      global bajada_broca=p[0,0,-0.012,0,0,0]
      $ 661 "bajada≔p[0,0,0.012,0,0,0]"
      global bajada=p[0,0,0.012,0,0,0]
      $ 662 "Direction: Base Z-"
      global move_thread_flag_662=0
      thread move_thread_662():
        enter_critical
        move_thread_flag_662 = 1
        local towardsPos=calculate_point_to_move_towards(p[0.0,0.0,0.0,0.0,0.0,0.0], [0.0,0.0,-1.0], 0.045)
        movel(towardsPos, a=0.025, v=0.02)
        move_thread_flag_662 = 2
        exit_critical
      end
      move_thread_flag_662 = 0
      move_thread_han_662 = run move_thread_662()
      while (True):
        sleep(1.0E-10)
        if (move_thread_flag_662 > 1):
          join move_thread_han_662
          $ 663 "Until (distance)"
          break
        end
        sync()
      end
      $ 664 "Popup: punto contacto alanzdo"
      popup("punto contacto alanzdo", "Mensaje", False, False, blocking=True)
      $ 665 "Direction: Base Z+"
      global move_thread_flag_665=0
      thread move_thread_665():
        enter_critical
        move_thread_flag_665 = 1
        local towardsPos=calculate_point_to_move_towards(p[0.0,0.0,0.0,0.0,0.0,0.0], [0.0,0.0,1.0], 0.001)
        movel(towardsPos, a=0.005, v=0.003)
        move_thread_flag_665 = 2
        exit_critical
      end
      move_thread_flag_665 = 0
      move_thread_han_665 = run move_thread_665()
      while (True):
        sleep(1.0E-10)
        if (move_thread_flag_665 > 1):
          join move_thread_han_665
          $ 666 "Until (distance)"
          break
        end
        sync()
      end
      $ 667 "Wait: 0.3"
      sleep(0.3)
      $ 668 "Set CO[1]=Encender"
      set_configurable_digital_out(1, True)
      $ 669 "Wait: 0.3"
      sleep(0.3)
      $ 670 "Loop 2 times"
      Loop_44 = 0
      while (Loop_44 < 2):
        $ 671 "bajar≔pose_add(get_actual_tcp_pose(), bajada_broca)"
        global bajar= pose_add ( get_actual_tcp_pose (), bajada_broca)
        $ 672 "bajar" "breakAfter"
        movel(bajar, a=0.005, v=0.001)
        $ 673 "subir≔pose_sub(get_actual_tcp_pose(), bajada_broca)"
        global subir= pose_sub ( get_actual_tcp_pose (), bajada_broca)
        $ 674 "subir" "breakAfter"
        movel(subir, a=0.01, v=0.005)
        $ 675 "bajada_broca≔pose_sub(bajada_broca, bajada)"
        global bajada_broca= pose_sub (bajada_broca, bajada)
        Loop_44 = Loop_44 + 1
      end
      $ 676 "Direction: Base Z+"
      global move_thread_flag_676=0
      thread move_thread_676():
        enter_critical
        move_thread_flag_676 = 1
        local towardsPos=calculate_point_to_move_towards(p[0.0,0.0,0.0,0.0,0.0,0.0], [0.0,0.0,1.0], 0.06)
        movel(towardsPos, a=0.035, v=0.03)
        move_thread_flag_676 = 2
        exit_critical
      end
      move_thread_flag_676 = 0
      move_thread_han_676 = run move_thread_676()
      while (True):
        sleep(1.0E-10)
        if (move_thread_flag_676 > 1):
          join move_thread_han_676
          $ 677 "Until (distance)"
          break
        end
        sync()
      end
      $ 678 "Set CO[1]=Apagar"
      set_configurable_digital_out(1, False)
      $ 679 "barreno_actual≔barreno_actual+1"
      global barreno_actual=barreno_actual+1
      $ 680 "If barreno_actual≥barrenos_menos1"
      if (barreno_actual >= barrenos_menos1):
        $ 681 "cambiar_broca≔ True "
        global cambiar_broca=  True
      end
      $ 682 "Call Quitar_broca"
      Quitar_broca()
      $ 683 "Call Poner_broca"
      Poner_broca()
    end
    $ 684 "Popup: Linea2 con full Terminada!"
    popup("Linea2 con full Terminada!", "Mensaje", False, False, blocking=True)
    $ 685 "Posicion3"
    $ 686 "eje7≔3"
    global eje7=3
    $ 687 "Broca_1"
    $ 688 "Linea3"
    $ 689 "Marcar_puntos"
    $ 690 "MoveL"
    $ 691 "Home3" "breakAfter"
    movel(Home3_p, a=0.5, v=0.1)
    $ 692 "Linea3_A" "breakAfter"
    movel(Linea3_A_p, a=0.5, v=0.1)
    $ 693 "Linea3_B" "breakAfter"
    movel(Linea3_B_p, a=0.5, v=0.1)
    $ 694 "Linea3_C" "breakAfter"
    movel(Linea3_C_p, a=0.5, v=0.1)
    $ 695 "Linea3_D" "breakAfter"
    movel(Linea3_D_p, a=0.5, v=0.1)
    $ 696 "Linea3_E" "breakAfter"
    movel(Linea3_E_p, a=0.5, v=0.1)
    $ 697 "Linea3_F" "breakAfter"
    movel(Linea3_F_p, a=0.5, v=0.1)
    $ 698 "AB"
    $ 699 "'desbaste_inicial'"
    # 'desbaste_inicial'
    $ 700 "bajada_broca≔p[0,0,-0.008,0,0,0]"
    global bajada_broca=p[0,0,-0.008,0,0,0]
    $ 701 "barrenos_menos1≔8"
    global barrenos_menos1=8
    $ 702 "barreno_actual≔0"
    global barreno_actual=0
    $ 703 "Loop barreno_actual≤barrenos_menos1"
    while (barreno_actual <= barrenos_menos1):
      $ 704 "Perforacion"
      $ 705 "MoveL"
      $ 706 "internos≔interpolate_pose(Linea3_A, Linea3_B, barreno_actual/barrenos_menos1)"
      global internos= interpolate_pose (Linea3_A_p, Linea3_B_p, barreno_actual/barrenos_menos1)
      $ 707 "internos" "breakAfter"
      movel(internos, a=0.5, v=0.1)
      $ 708 "'desbaste_inicial'"
      # 'desbaste_inicial'
      $ 709 "bajada_broca≔p[0,0,-0.008,0,0,0]"
      global bajada_broca=p[0,0,-0.008,0,0,0]
      $ 710 "bajada≔p[0,0,0.008,0,0,0]"
      global bajada=p[0,0,0.008,0,0,0]
      $ 711 "Direction: Base Z-"
      global move_thread_flag_711=0
      thread move_thread_711():
        enter_critical
        move_thread_flag_711 = 1
        local towardsPos=calculate_point_to_move_towards(p[0.0,0.0,0.0,0.0,0.0,0.0], [0.0,0.0,-1.0], 0.055)
        movel(towardsPos, a=0.015, v=0.02)
        move_thread_flag_711 = 2
        exit_critical
      end
      move_thread_flag_711 = 0
      move_thread_han_711 = run move_thread_711()
      while (True):
        sleep(1.0E-10)
        if (move_thread_flag_711 > 1):
          join move_thread_han_711
          $ 712 "Until (distance)"
          break
        end
        sync()
      end
      $ 713 "Popup: punto contacto alanzdo"
      popup("punto contacto alanzdo", "Mensaje", False, False, blocking=True)
      $ 714 "Direction: Base Z+"
      global move_thread_flag_714=0
      thread move_thread_714():
        enter_critical
        move_thread_flag_714 = 1
        local towardsPos=calculate_point_to_move_towards(p[0.0,0.0,0.0,0.0,0.0,0.0], [0.0,0.0,1.0], 0.002)
        movel(towardsPos, a=0.005, v=0.003)
        move_thread_flag_714 = 2
        exit_critical
      end
      move_thread_flag_714 = 0
      move_thread_han_714 = run move_thread_714()
      while (True):
        sleep(1.0E-10)
        if (move_thread_flag_714 > 1):
          join move_thread_han_714
          $ 715 "Until (distance)"
          break
        end
        sync()
      end
      $ 716 "Wait: 0.3"
      sleep(0.3)
      $ 717 "Set CO[1]=Encender"
      set_configurable_digital_out(1, True)
      $ 718 "Wait: 0.3"
      sleep(0.3)
      $ 719 "Loop 3 times"
      Loop_3 = 0
      while (Loop_3 < 3):
        $ 720 "bajar≔pose_add(get_actual_tcp_pose(), bajada_broca)"
        global bajar= pose_add ( get_actual_tcp_pose (), bajada_broca)
        $ 721 "bajar" "breakAfter"
        movel(bajar, a=0.005, v=0.001)
        $ 722 "subir≔pose_sub(get_actual_tcp_pose(), bajada_broca)"
        global subir= pose_sub ( get_actual_tcp_pose (), bajada_broca)
        $ 723 "subir" "breakAfter"
        movel(subir, a=0.01, v=0.01)
        $ 724 "bajada_broca≔pose_sub(bajada_broca, bajada)"
        global bajada_broca= pose_sub (bajada_broca, bajada)
        Loop_3 = Loop_3 + 1
      end
      $ 725 "Direction: Base Z+"
      global move_thread_flag_725=0
      thread move_thread_725():
        enter_critical
        move_thread_flag_725 = 1
        local towardsPos=calculate_point_to_move_towards(p[0.0,0.0,0.0,0.0,0.0,0.0], [0.0,0.0,1.0], 0.06)
        movel(towardsPos, a=0.035, v=0.03)
        move_thread_flag_725 = 2
        exit_critical
      end
      move_thread_flag_725 = 0
      move_thread_han_725 = run move_thread_725()
      while (True):
        sleep(1.0E-10)
        if (move_thread_flag_725 > 1):
          join move_thread_han_725
          $ 726 "Until (distance)"
          break
        end
        sync()
      end
      $ 727 "Set CO[1]=Apagar"
      set_configurable_digital_out(1, False)
      $ 728 "barreno_actual≔barreno_actual+1"
      global barreno_actual=barreno_actual+1
    end
    $ 731 "CD"
    $ 732 "'desbaste_inicial'"
    # 'desbaste_inicial'
    $ 733 "bajada_broca≔p[0,0,-0.008,0,0,0]"
    global bajada_broca=p[0,0,-0.008,0,0,0]
    $ 734 "barrenos_menos1≔8"
    global barrenos_menos1=8
    $ 735 "barreno_actual≔0"
    global barreno_actual=0
    $ 736 "Loop barreno_actual≤barrenos_menos1"
    while (barreno_actual <= barrenos_menos1):
      $ 737 "Perforacion"
      $ 738 "MoveL"
      $ 739 "internos≔interpolate_pose(Linea3_C, Linea3_D, barreno_actual/barrenos_menos1)"
      global internos= interpolate_pose (Linea3_C_p, Linea3_D_p, barreno_actual/barrenos_menos1)
      $ 740 "internos" "breakAfter"
      movel(internos, a=0.5, v=0.1)
      $ 741 "'desbaste_inicial'"
      # 'desbaste_inicial'
      $ 742 "bajada_broca≔p[0,0,-0.008,0,0,0]"
      global bajada_broca=p[0,0,-0.008,0,0,0]
      $ 743 "bajada≔p[0,0,0.008,0,0,0]"
      global bajada=p[0,0,0.008,0,0,0]
      $ 744 "Direction: Base Z-"
      global move_thread_flag_744=0
      thread move_thread_744():
        enter_critical
        move_thread_flag_744 = 1
        local towardsPos=calculate_point_to_move_towards(p[0.0,0.0,0.0,0.0,0.0,0.0], [0.0,0.0,-1.0], 0.055)
        movel(towardsPos, a=0.015, v=0.02)
        move_thread_flag_744 = 2
        exit_critical
      end
      move_thread_flag_744 = 0
      move_thread_han_744 = run move_thread_744()
      while (True):
        sleep(1.0E-10)
        if (move_thread_flag_744 > 1):
          join move_thread_han_744
          $ 745 "Until (distance)"
          break
        end
        sync()
      end
      $ 746 "Popup: punto contacto alanzdo"
      popup("punto contacto alanzdo", "Mensaje", False, False, blocking=True)
      $ 747 "Direction: Base Z+"
      global move_thread_flag_747=0
      thread move_thread_747():
        enter_critical
        move_thread_flag_747 = 1
        local towardsPos=calculate_point_to_move_towards(p[0.0,0.0,0.0,0.0,0.0,0.0], [0.0,0.0,1.0], 0.002)
        movel(towardsPos, a=0.005, v=0.003)
        move_thread_flag_747 = 2
        exit_critical
      end
      move_thread_flag_747 = 0
      move_thread_han_747 = run move_thread_747()
      while (True):
        sleep(1.0E-10)
        if (move_thread_flag_747 > 1):
          join move_thread_han_747
          $ 748 "Until (distance)"
          break
        end
        sync()
      end
      $ 749 "Wait: 0.3"
      sleep(0.3)
      $ 750 "Set CO[1]=Encender"
      set_configurable_digital_out(1, True)
      $ 751 "Wait: 0.3"
      sleep(0.3)
      $ 752 "Loop 3 times"
      Loop_6 = 0
      while (Loop_6 < 3):
        $ 753 "bajar≔pose_add(get_actual_tcp_pose(), bajada_broca)"
        global bajar= pose_add ( get_actual_tcp_pose (), bajada_broca)
        $ 754 "bajar" "breakAfter"
        movel(bajar, a=0.005, v=0.001)
        $ 755 "subir≔pose_sub(get_actual_tcp_pose(), bajada_broca)"
        global subir= pose_sub ( get_actual_tcp_pose (), bajada_broca)
        $ 756 "subir" "breakAfter"
        movel(subir, a=0.01, v=0.01)
        $ 757 "bajada_broca≔pose_sub(bajada_broca, bajada)"
        global bajada_broca= pose_sub (bajada_broca, bajada)
        Loop_6 = Loop_6 + 1
      end
      $ 758 "Direction: Base Z+"
      global move_thread_flag_758=0
      thread move_thread_758():
        enter_critical
        move_thread_flag_758 = 1
        local towardsPos=calculate_point_to_move_towards(p[0.0,0.0,0.0,0.0,0.0,0.0], [0.0,0.0,1.0], 0.06)
        movel(towardsPos, a=0.035, v=0.03)
        move_thread_flag_758 = 2
        exit_critical
      end
      move_thread_flag_758 = 0
      move_thread_han_758 = run move_thread_758()
      while (True):
        sleep(1.0E-10)
        if (move_thread_flag_758 > 1):
          join move_thread_han_758
          $ 759 "Until (distance)"
          break
        end
        sync()
      end
      $ 760 "Set CO[1]=Apagar"
      set_configurable_digital_out(1, False)
      $ 761 "barreno_actual≔barreno_actual+1"
      global barreno_actual=barreno_actual+1
    end
    $ 764 "EF"
    $ 765 "'desbaste_inicial'"
    # 'desbaste_inicial'
    $ 766 "bajada_broca≔p[0,0,-0.008,0,0,0]"
    global bajada_broca=p[0,0,-0.008,0,0,0]
    $ 767 "barrenos_menos1≔8"
    global barrenos_menos1=8
    $ 768 "barreno_actual≔0"
    global barreno_actual=0
    $ 769 "Loop barreno_actual≤barrenos_menos1"
    while (barreno_actual <= barrenos_menos1):
      $ 770 "Perforacion"
      $ 771 "MoveL"
      $ 772 "internos≔interpolate_pose(Linea3_E, Linea3_F, barreno_actual/barrenos_menos1)"
      global internos= interpolate_pose (Linea3_E_p, Linea3_F_p, barreno_actual/barrenos_menos1)
      $ 773 "internos" "breakAfter"
      movel(internos, a=0.5, v=0.1)
      $ 774 "'desbaste_inicial'"
      # 'desbaste_inicial'
      $ 775 "bajada_broca≔p[0,0,-0.008,0,0,0]"
      global bajada_broca=p[0,0,-0.008,0,0,0]
      $ 776 "bajada≔p[0,0,0.008,0,0,0]"
      global bajada=p[0,0,0.008,0,0,0]
      $ 777 "Direction: Base Z-"
      global move_thread_flag_777=0
      thread move_thread_777():
        enter_critical
        move_thread_flag_777 = 1
        local towardsPos=calculate_point_to_move_towards(p[0.0,0.0,0.0,0.0,0.0,0.0], [0.0,0.0,-1.0], 0.055)
        movel(towardsPos, a=0.015, v=0.02)
        move_thread_flag_777 = 2
        exit_critical
      end
      move_thread_flag_777 = 0
      move_thread_han_777 = run move_thread_777()
      while (True):
        sleep(1.0E-10)
        if (move_thread_flag_777 > 1):
          join move_thread_han_777
          $ 778 "Until (distance)"
          break
        end
        sync()
      end
      $ 779 "Popup: punto contacto alanzdo"
      popup("punto contacto alanzdo", "Mensaje", False, False, blocking=True)
      $ 780 "Direction: Base Z+"
      global move_thread_flag_780=0
      thread move_thread_780():
        enter_critical
        move_thread_flag_780 = 1
        local towardsPos=calculate_point_to_move_towards(p[0.0,0.0,0.0,0.0,0.0,0.0], [0.0,0.0,1.0], 0.002)
        movel(towardsPos, a=0.005, v=0.003)
        move_thread_flag_780 = 2
        exit_critical
      end
      move_thread_flag_780 = 0
      move_thread_han_780 = run move_thread_780()
      while (True):
        sleep(1.0E-10)
        if (move_thread_flag_780 > 1):
          join move_thread_han_780
          $ 781 "Until (distance)"
          break
        end
        sync()
      end
      $ 782 "Wait: 0.3"
      sleep(0.3)
      $ 783 "Set CO[1]=Encender"
      set_configurable_digital_out(1, True)
      $ 784 "Wait: 0.3"
      sleep(0.3)
      $ 785 "Loop 3 times"
      Loop_8 = 0
      while (Loop_8 < 3):
        $ 786 "bajar≔pose_add(get_actual_tcp_pose(), bajada_broca)"
        global bajar= pose_add ( get_actual_tcp_pose (), bajada_broca)
        $ 787 "bajar" "breakAfter"
        movel(bajar, a=0.005, v=0.001)
        $ 788 "subir≔pose_sub(get_actual_tcp_pose(), bajada_broca)"
        global subir= pose_sub ( get_actual_tcp_pose (), bajada_broca)
        $ 789 "subir" "breakAfter"
        movel(subir, a=0.01, v=0.01)
        $ 790 "bajada_broca≔pose_sub(bajada_broca, bajada)"
        global bajada_broca= pose_sub (bajada_broca, bajada)
        Loop_8 = Loop_8 + 1
      end
      $ 791 "Direction: Base Z+"
      global move_thread_flag_791=0
      thread move_thread_791():
        enter_critical
        move_thread_flag_791 = 1
        local towardsPos=calculate_point_to_move_towards(p[0.0,0.0,0.0,0.0,0.0,0.0], [0.0,0.0,1.0], 0.06)
        movel(towardsPos, a=0.035, v=0.03)
        move_thread_flag_791 = 2
        exit_critical
      end
      move_thread_flag_791 = 0
      move_thread_han_791 = run move_thread_791()
      while (True):
        sleep(1.0E-10)
        if (move_thread_flag_791 > 1):
          join move_thread_han_791
          $ 792 "Until (distance)"
          break
        end
        sync()
      end
      $ 793 "Set CO[1]=Apagar"
      set_configurable_digital_out(1, False)
      $ 794 "barreno_actual≔barreno_actual+1"
      global barreno_actual=barreno_actual+1
    end
    $ 797 "Popup: Linea3 con chica Terminada!"
    popup("Linea3 con chica Terminada!", "Mensaje", False, False, blocking=True)
    $ 798 "Linea4"
    $ 799 "Marcar_puntos"
    $ 800 "MoveL"
    $ 801 "Home3" "breakAfter"
    movel(Home3_p, a=0.5, v=0.1)
    $ 802 "Linea4_A" "breakAfter"
    movel(Linea4_A_p, a=0.5, v=0.1)
    $ 803 "Linea4_B" "breakAfter"
    movel(Linea4_B_p, a=0.5, v=0.1)
    $ 804 "Linea4_C" "breakAfter"
    movel(Linea4_C_p, a=0.5, v=0.1)
    $ 805 "Linea4_D" "breakAfter"
    movel(Linea4_D_p, a=0.5, v=0.1)
    $ 806 "Linea4_E" "breakAfter"
    movel(Linea4_E_p, a=0.5, v=0.1)
    $ 807 "Linea4_F" "breakAfter"
    movel(Linea4_F_p, a=0.5, v=0.1)
    $ 808 "AB"
    $ 809 "'desbaste_inicial'"
    # 'desbaste_inicial'
    $ 810 "bajada_broca≔p[0,0,-0.008,0,0,0]"
    global bajada_broca=p[0,0,-0.008,0,0,0]
    $ 811 "barrenos_menos1≔8"
    global barrenos_menos1=8
    $ 812 "barreno_actual≔0"
    global barreno_actual=0
    $ 813 "Loop barreno_actual≤barrenos_menos1"
    while (barreno_actual <= barrenos_menos1):
      $ 814 "Perforacion"
      $ 815 "MoveL"
      $ 816 "internos≔interpolate_pose(Linea4_A, Linea4_B, barreno_actual/barrenos_menos1)"
      global internos= interpolate_pose (Linea4_A_p, Linea4_B_p, barreno_actual/barrenos_menos1)
      $ 817 "internos" "breakAfter"
      movel(internos, a=0.5, v=0.1)
      $ 818 "'desbaste_inicial'"
      # 'desbaste_inicial'
      $ 819 "bajada_broca≔p[0,0,-0.008,0,0,0]"
      global bajada_broca=p[0,0,-0.008,0,0,0]
      $ 820 "bajada≔p[0,0,0.008,0,0,0]"
      global bajada=p[0,0,0.008,0,0,0]
      $ 821 "Direction: Base Z-"
      global move_thread_flag_821=0
      thread move_thread_821():
        enter_critical
        move_thread_flag_821 = 1
        local towardsPos=calculate_point_to_move_towards(p[0.0,0.0,0.0,0.0,0.0,0.0], [0.0,0.0,-1.0], 0.055)
        movel(towardsPos, a=0.015, v=0.02)
        move_thread_flag_821 = 2
        exit_critical
      end
      move_thread_flag_821 = 0
      move_thread_han_821 = run move_thread_821()
      while (True):
        sleep(1.0E-10)
        if (move_thread_flag_821 > 1):
          join move_thread_han_821
          $ 822 "Until (distance)"
          break
        end
        sync()
      end
      $ 823 "Popup: punto contacto alanzdo"
      popup("punto contacto alanzdo", "Mensaje", False, False, blocking=True)
      $ 824 "Direction: Base Z+"
      global move_thread_flag_824=0
      thread move_thread_824():
        enter_critical
        move_thread_flag_824 = 1
        local towardsPos=calculate_point_to_move_towards(p[0.0,0.0,0.0,0.0,0.0,0.0], [0.0,0.0,1.0], 0.002)
        movel(towardsPos, a=0.005, v=0.003)
        move_thread_flag_824 = 2
        exit_critical
      end
      move_thread_flag_824 = 0
      move_thread_han_824 = run move_thread_824()
      while (True):
        sleep(1.0E-10)
        if (move_thread_flag_824 > 1):
          join move_thread_han_824
          $ 825 "Until (distance)"
          break
        end
        sync()
      end
      $ 826 "Wait: 0.3"
      sleep(0.3)
      $ 827 "Set CO[1]=Encender"
      set_configurable_digital_out(1, True)
      $ 828 "Wait: 0.3"
      sleep(0.3)
      $ 829 "Loop 3 times"
      Loop_12 = 0
      while (Loop_12 < 3):
        $ 830 "bajar≔pose_add(get_actual_tcp_pose(), bajada_broca)"
        global bajar= pose_add ( get_actual_tcp_pose (), bajada_broca)
        $ 831 "bajar" "breakAfter"
        movel(bajar, a=0.005, v=0.001)
        $ 832 "subir≔pose_sub(get_actual_tcp_pose(), bajada_broca)"
        global subir= pose_sub ( get_actual_tcp_pose (), bajada_broca)
        $ 833 "subir" "breakAfter"
        movel(subir, a=0.01, v=0.01)
        $ 834 "bajada_broca≔pose_sub(bajada_broca, bajada)"
        global bajada_broca= pose_sub (bajada_broca, bajada)
        Loop_12 = Loop_12 + 1
      end
      $ 835 "Direction: Base Z+"
      global move_thread_flag_835=0
      thread move_thread_835():
        enter_critical
        move_thread_flag_835 = 1
        local towardsPos=calculate_point_to_move_towards(p[0.0,0.0,0.0,0.0,0.0,0.0], [0.0,0.0,1.0], 0.06)
        movel(towardsPos, a=0.035, v=0.03)
        move_thread_flag_835 = 2
        exit_critical
      end
      move_thread_flag_835 = 0
      move_thread_han_835 = run move_thread_835()
      while (True):
        sleep(1.0E-10)
        if (move_thread_flag_835 > 1):
          join move_thread_han_835
          $ 836 "Until (distance)"
          break
        end
        sync()
      end
      $ 837 "Set CO[1]=Apagar"
      set_configurable_digital_out(1, False)
      $ 838 "barreno_actual≔barreno_actual+1"
      global barreno_actual=barreno_actual+1
    end
    $ 841 "CD"
    $ 842 "'desbaste_inicial'"
    # 'desbaste_inicial'
    $ 843 "bajada_broca≔p[0,0,-0.008,0,0,0]"
    global bajada_broca=p[0,0,-0.008,0,0,0]
    $ 844 "barrenos_menos1≔8"
    global barrenos_menos1=8
    $ 845 "barreno_actual≔0"
    global barreno_actual=0
    $ 846 "Loop barreno_actual≤barrenos_menos1"
    while (barreno_actual <= barrenos_menos1):
      $ 847 "Perforacion"
      $ 848 "MoveL"
      $ 849 "internos≔interpolate_pose(Linea4_C, Linea4_D, barreno_actual/barrenos_menos1)"
      global internos= interpolate_pose (Linea4_C_p, Linea4_D_p, barreno_actual/barrenos_menos1)
      $ 850 "internos" "breakAfter"
      movel(internos, a=0.5, v=0.1)
      $ 851 "'desbaste_inicial'"
      # 'desbaste_inicial'
      $ 852 "bajada_broca≔p[0,0,-0.008,0,0,0]"
      global bajada_broca=p[0,0,-0.008,0,0,0]
      $ 853 "bajada≔p[0,0,0.008,0,0,0]"
      global bajada=p[0,0,0.008,0,0,0]
      $ 854 "Direction: Base Z-"
      global move_thread_flag_854=0
      thread move_thread_854():
        enter_critical
        move_thread_flag_854 = 1
        local towardsPos=calculate_point_to_move_towards(p[0.0,0.0,0.0,0.0,0.0,0.0], [0.0,0.0,-1.0], 0.055)
        movel(towardsPos, a=0.015, v=0.02)
        move_thread_flag_854 = 2
        exit_critical
      end
      move_thread_flag_854 = 0
      move_thread_han_854 = run move_thread_854()
      while (True):
        sleep(1.0E-10)
        if (move_thread_flag_854 > 1):
          join move_thread_han_854
          $ 855 "Until (distance)"
          break
        end
        sync()
      end
      $ 856 "Popup: punto contacto alanzdo"
      popup("punto contacto alanzdo", "Mensaje", False, False, blocking=True)
      $ 857 "Direction: Base Z+"
      global move_thread_flag_857=0
      thread move_thread_857():
        enter_critical
        move_thread_flag_857 = 1
        local towardsPos=calculate_point_to_move_towards(p[0.0,0.0,0.0,0.0,0.0,0.0], [0.0,0.0,1.0], 0.002)
        movel(towardsPos, a=0.005, v=0.003)
        move_thread_flag_857 = 2
        exit_critical
      end
      move_thread_flag_857 = 0
      move_thread_han_857 = run move_thread_857()
      while (True):
        sleep(1.0E-10)
        if (move_thread_flag_857 > 1):
          join move_thread_han_857
          $ 858 "Until (distance)"
          break
        end
        sync()
      end
      $ 859 "Wait: 0.3"
      sleep(0.3)
      $ 860 "Set CO[1]=Encender"
      set_configurable_digital_out(1, True)
      $ 861 "Wait: 0.3"
      sleep(0.3)
      $ 862 "Loop 3 times"
      Loop_15 = 0
      while (Loop_15 < 3):
        $ 863 "bajar≔pose_add(get_actual_tcp_pose(), bajada_broca)"
        global bajar= pose_add ( get_actual_tcp_pose (), bajada_broca)
        $ 864 "bajar" "breakAfter"
        movel(bajar, a=0.005, v=0.001)
        $ 865 "subir≔pose_sub(get_actual_tcp_pose(), bajada_broca)"
        global subir= pose_sub ( get_actual_tcp_pose (), bajada_broca)
        $ 866 "subir" "breakAfter"
        movel(subir, a=0.01, v=0.01)
        $ 867 "bajada_broca≔pose_sub(bajada_broca, bajada)"
        global bajada_broca= pose_sub (bajada_broca, bajada)
        Loop_15 = Loop_15 + 1
      end
      $ 868 "Direction: Base Z+"
      global move_thread_flag_868=0
      thread move_thread_868():
        enter_critical
        move_thread_flag_868 = 1
        local towardsPos=calculate_point_to_move_towards(p[0.0,0.0,0.0,0.0,0.0,0.0], [0.0,0.0,1.0], 0.06)
        movel(towardsPos, a=0.035, v=0.03)
        move_thread_flag_868 = 2
        exit_critical
      end
      move_thread_flag_868 = 0
      move_thread_han_868 = run move_thread_868()
      while (True):
        sleep(1.0E-10)
        if (move_thread_flag_868 > 1):
          join move_thread_han_868
          $ 869 "Until (distance)"
          break
        end
        sync()
      end
      $ 870 "Set CO[1]=Apagar"
      set_configurable_digital_out(1, False)
      $ 871 "barreno_actual≔barreno_actual+1"
      global barreno_actual=barreno_actual+1
    end
    $ 874 "EF"
    $ 875 "'desbaste_inicial'"
    # 'desbaste_inicial'
    $ 876 "bajada_broca≔p[0,0,-0.008,0,0,0]"
    global bajada_broca=p[0,0,-0.008,0,0,0]
    $ 877 "barrenos_menos1≔8"
    global barrenos_menos1=8
    $ 878 "barreno_actual≔0"
    global barreno_actual=0
    $ 879 "Loop barreno_actual≤barrenos_menos1"
    while (barreno_actual <= barrenos_menos1):
      $ 880 "Perforacion"
      $ 881 "MoveL"
      $ 882 "internos≔interpolate_pose(Linea4_E, Linea4_F, barreno_actual/barrenos_menos1)"
      global internos= interpolate_pose (Linea4_E_p, Linea4_F_p, barreno_actual/barrenos_menos1)
      $ 883 "internos" "breakAfter"
      movel(internos, a=0.5, v=0.1)
      $ 884 "'desbaste_inicial'"
      # 'desbaste_inicial'
      $ 885 "bajada_broca≔p[0,0,-0.008,0,0,0]"
      global bajada_broca=p[0,0,-0.008,0,0,0]
      $ 886 "bajada≔p[0,0,0.008,0,0,0]"
      global bajada=p[0,0,0.008,0,0,0]
      $ 887 "Direction: Base Z-"
      global move_thread_flag_887=0
      thread move_thread_887():
        enter_critical
        move_thread_flag_887 = 1
        local towardsPos=calculate_point_to_move_towards(p[0.0,0.0,0.0,0.0,0.0,0.0], [0.0,0.0,-1.0], 0.055)
        movel(towardsPos, a=0.015, v=0.02)
        move_thread_flag_887 = 2
        exit_critical
      end
      move_thread_flag_887 = 0
      move_thread_han_887 = run move_thread_887()
      while (True):
        sleep(1.0E-10)
        if (move_thread_flag_887 > 1):
          join move_thread_han_887
          $ 888 "Until (distance)"
          break
        end
        sync()
      end
      $ 889 "Popup: punto contacto alanzdo"
      popup("punto contacto alanzdo", "Mensaje", False, False, blocking=True)
      $ 890 "Direction: Base Z+"
      global move_thread_flag_890=0
      thread move_thread_890():
        enter_critical
        move_thread_flag_890 = 1
        local towardsPos=calculate_point_to_move_towards(p[0.0,0.0,0.0,0.0,0.0,0.0], [0.0,0.0,1.0], 0.002)
        movel(towardsPos, a=0.005, v=0.003)
        move_thread_flag_890 = 2
        exit_critical
      end
      move_thread_flag_890 = 0
      move_thread_han_890 = run move_thread_890()
      while (True):
        sleep(1.0E-10)
        if (move_thread_flag_890 > 1):
          join move_thread_han_890
          $ 891 "Until (distance)"
          break
        end
        sync()
      end
      $ 892 "Wait: 0.3"
      sleep(0.3)
      $ 893 "Set CO[1]=Encender"
      set_configurable_digital_out(1, True)
      $ 894 "Wait: 0.3"
      sleep(0.3)
      $ 895 "Loop 3 times"
      Loop_19 = 0
      while (Loop_19 < 3):
        $ 896 "bajar≔pose_add(get_actual_tcp_pose(), bajada_broca)"
        global bajar= pose_add ( get_actual_tcp_pose (), bajada_broca)
        $ 897 "bajar" "breakAfter"
        movel(bajar, a=0.005, v=0.001)
        $ 898 "subir≔pose_sub(get_actual_tcp_pose(), bajada_broca)"
        global subir= pose_sub ( get_actual_tcp_pose (), bajada_broca)
        $ 899 "subir" "breakAfter"
        movel(subir, a=0.01, v=0.01)
        $ 900 "bajada_broca≔pose_sub(bajada_broca, bajada)"
        global bajada_broca= pose_sub (bajada_broca, bajada)
        Loop_19 = Loop_19 + 1
      end
      $ 901 "Direction: Base Z+"
      global move_thread_flag_901=0
      thread move_thread_901():
        enter_critical
        move_thread_flag_901 = 1
        local towardsPos=calculate_point_to_move_towards(p[0.0,0.0,0.0,0.0,0.0,0.0], [0.0,0.0,1.0], 0.06)
        movel(towardsPos, a=0.035, v=0.03)
        move_thread_flag_901 = 2
        exit_critical
      end
      move_thread_flag_901 = 0
      move_thread_han_901 = run move_thread_901()
      while (True):
        sleep(1.0E-10)
        if (move_thread_flag_901 > 1):
          join move_thread_han_901
          $ 902 "Until (distance)"
          break
        end
        sync()
      end
      $ 903 "Set CO[1]=Apagar"
      set_configurable_digital_out(1, False)
      $ 904 "barreno_actual≔barreno_actual+1"
      global barreno_actual=barreno_actual+1
      $ 905 "If barreno_actual≥barrenos_menos1"
      if (barreno_actual >= barrenos_menos1):
        $ 906 "cambiar_broca≔ True "
        global cambiar_broca=  True
      end
    end
    $ 909 "Popup: Linea4 con chica Terminada!"
    popup("Linea4 con chica Terminada!", "Mensaje", False, False, blocking=True)
    $ 910 "Broca_2"
    $ 911 "Linea3"
    $ 912 "Marcar_puntos"
    $ 913 "MoveL"
    $ 914 "Home3" "breakAfter"
    movel(Home3_p, a=0.5, v=0.1)
    $ 915 "Linea3_A" "breakAfter"
    movel(Linea3_A_p, a=0.5, v=0.1)
    $ 916 "Linea3_B" "breakAfter"
    movel(Linea3_B_p, a=0.5, v=0.1)
    $ 917 "Linea3_C" "breakAfter"
    movel(Linea3_C_p, a=0.5, v=0.1)
    $ 918 "Linea3_D" "breakAfter"
    movel(Linea3_D_p, a=0.5, v=0.1)
    $ 919 "Linea3_E" "breakAfter"
    movel(Linea3_E_p, a=0.5, v=0.1)
    $ 920 "Linea3_F" "breakAfter"
    movel(Linea3_F_p, a=0.5, v=0.1)
    $ 921 "AB"
    $ 922 "'desbaste_inicial'"
    # 'desbaste_inicial'
    $ 923 "bajada_broca≔p[0,0,-0.012,0,0,0]"
    global bajada_broca=p[0,0,-0.012,0,0,0]
    $ 924 "barrenos_menos1≔8"
    global barrenos_menos1=8
    $ 925 "barreno_actual≔0"
    global barreno_actual=0
    $ 926 "Loop barreno_actual≤barrenos_menos1"
    while (barreno_actual <= barrenos_menos1):
      $ 927 "Perforacion"
      $ 928 "MoveL"
      $ 929 "internos≔interpolate_pose(Linea3_A, Linea3_B, barreno_actual/barrenos_menos1)"
      global internos= interpolate_pose (Linea3_A_p, Linea3_B_p, barreno_actual/barrenos_menos1)
      $ 930 "internos" "breakAfter"
      movel(internos, a=0.5, v=0.1)
      $ 931 "'desbaste_inicial'"
      # 'desbaste_inicial'
      $ 932 "bajada_broca≔p[0,0,-0.012,0,0,0]"
      global bajada_broca=p[0,0,-0.012,0,0,0]
      $ 933 "bajada≔p[0,0,0.012,0,0,0]"
      global bajada=p[0,0,0.012,0,0,0]
      $ 934 "Direction: Base Z-"
      global move_thread_flag_934=0
      thread move_thread_934():
        enter_critical
        move_thread_flag_934 = 1
        local towardsPos=calculate_point_to_move_towards(p[0.0,0.0,0.0,0.0,0.0,0.0], [0.0,0.0,-1.0], 0.055)
        movel(towardsPos, a=0.015, v=0.02)
        move_thread_flag_934 = 2
        exit_critical
      end
      move_thread_flag_934 = 0
      move_thread_han_934 = run move_thread_934()
      while (True):
        sleep(1.0E-10)
        if (move_thread_flag_934 > 1):
          join move_thread_han_934
          $ 935 "Until (distance)"
          break
        end
        sync()
      end
      $ 936 "Popup: punto contacto alanzdo"
      popup("punto contacto alanzdo", "Mensaje", False, False, blocking=True)
      $ 937 "Direction: Base Z+"
      global move_thread_flag_937=0
      thread move_thread_937():
        enter_critical
        move_thread_flag_937 = 1
        local towardsPos=calculate_point_to_move_towards(p[0.0,0.0,0.0,0.0,0.0,0.0], [0.0,0.0,1.0], 0.001)
        movel(towardsPos, a=0.005, v=0.003)
        move_thread_flag_937 = 2
        exit_critical
      end
      move_thread_flag_937 = 0
      move_thread_han_937 = run move_thread_937()
      while (True):
        sleep(1.0E-10)
        if (move_thread_flag_937 > 1):
          join move_thread_han_937
          $ 938 "Until (distance)"
          break
        end
        sync()
      end
      $ 939 "Wait: 0.3"
      sleep(0.3)
      $ 940 "Set CO[1]=Encender"
      set_configurable_digital_out(1, True)
      $ 941 "Wait: 0.3"
      sleep(0.3)
      $ 942 "Loop 2 times"
      Loop_23 = 0
      while (Loop_23 < 2):
        $ 943 "bajar≔pose_add(get_actual_tcp_pose(), bajada_broca)"
        global bajar= pose_add ( get_actual_tcp_pose (), bajada_broca)
        $ 944 "bajar" "breakAfter"
        movel(bajar, a=0.005, v=0.001)
        $ 945 "subir≔pose_sub(get_actual_tcp_pose(), bajada_broca)"
        global subir= pose_sub ( get_actual_tcp_pose (), bajada_broca)
        $ 946 "subir" "breakAfter"
        movel(subir, a=0.01, v=0.01)
        $ 947 "bajada_broca≔pose_sub(bajada_broca, bajada)"
        global bajada_broca= pose_sub (bajada_broca, bajada)
        Loop_23 = Loop_23 + 1
      end
      $ 948 "Direction: Base Z+"
      global move_thread_flag_948=0
      thread move_thread_948():
        enter_critical
        move_thread_flag_948 = 1
        local towardsPos=calculate_point_to_move_towards(p[0.0,0.0,0.0,0.0,0.0,0.0], [0.0,0.0,1.0], 0.06)
        movel(towardsPos, a=0.035, v=0.03)
        move_thread_flag_948 = 2
        exit_critical
      end
      move_thread_flag_948 = 0
      move_thread_han_948 = run move_thread_948()
      while (True):
        sleep(1.0E-10)
        if (move_thread_flag_948 > 1):
          join move_thread_han_948
          $ 949 "Until (distance)"
          break
        end
        sync()
      end
      $ 950 "Set CO[1]=Apagar"
      set_configurable_digital_out(1, False)
      $ 951 "barreno_actual≔barreno_actual+1"
      global barreno_actual=barreno_actual+1
    end
    $ 954 "CD"
    $ 955 "'desbaste_inicial'"
    # 'desbaste_inicial'
    $ 956 "bajada_broca≔p[0,0,-0.012,0,0,0]"
    global bajada_broca=p[0,0,-0.012,0,0,0]
    $ 957 "barrenos_menos1≔8"
    global barrenos_menos1=8
    $ 958 "barreno_actual≔0"
    global barreno_actual=0
    $ 959 "Loop barreno_actual≤barrenos_menos1"
    while (barreno_actual <= barrenos_menos1):
      $ 960 "Perforacion"
      $ 961 "MoveL"
      $ 962 "internos≔interpolate_pose(Linea3_C, Linea3_D, barreno_actual/barrenos_menos1)"
      global internos= interpolate_pose (Linea3_C_p, Linea3_D_p, barreno_actual/barrenos_menos1)
      $ 963 "internos" "breakAfter"
      movel(internos, a=0.5, v=0.1)
      $ 964 "'desbaste_inicial'"
      # 'desbaste_inicial'
      $ 965 "bajada_broca≔p[0,0,-0.012,0,0,0]"
      global bajada_broca=p[0,0,-0.012,0,0,0]
      $ 966 "bajada≔p[0,0,0.012,0,0,0]"
      global bajada=p[0,0,0.012,0,0,0]
      $ 967 "Direction: Base Z-"
      global move_thread_flag_967=0
      thread move_thread_967():
        enter_critical
        move_thread_flag_967 = 1
        local towardsPos=calculate_point_to_move_towards(p[0.0,0.0,0.0,0.0,0.0,0.0], [0.0,0.0,-1.0], 0.055)
        movel(towardsPos, a=0.015, v=0.02)
        move_thread_flag_967 = 2
        exit_critical
      end
      move_thread_flag_967 = 0
      move_thread_han_967 = run move_thread_967()
      while (True):
        sleep(1.0E-10)
        if (move_thread_flag_967 > 1):
          join move_thread_han_967
          $ 968 "Until (distance)"
          break
        end
        sync()
      end
      $ 969 "Popup: punto contacto alanzdo"
      popup("punto contacto alanzdo", "Mensaje", False, False, blocking=True)
      $ 970 "Direction: Base Z+"
      global move_thread_flag_970=0
      thread move_thread_970():
        enter_critical
        move_thread_flag_970 = 1
        local towardsPos=calculate_point_to_move_towards(p[0.0,0.0,0.0,0.0,0.0,0.0], [0.0,0.0,1.0], 0.001)
        movel(towardsPos, a=0.005, v=0.003)
        move_thread_flag_970 = 2
        exit_critical
      end
      move_thread_flag_970 = 0
      move_thread_han_970 = run move_thread_970()
      while (True):
        sleep(1.0E-10)
        if (move_thread_flag_970 > 1):
          join move_thread_han_970
          $ 971 "Until (distance)"
          break
        end
        sync()
      end
      $ 972 "Wait: 0.3"
      sleep(0.3)
      $ 973 "Set CO[1]=Encender"
      set_configurable_digital_out(1, True)
      $ 974 "Wait: 0.3"
      sleep(0.3)
      $ 975 "Loop 2 times"
      Loop_25 = 0
      while (Loop_25 < 2):
        $ 976 "bajar≔pose_add(get_actual_tcp_pose(), bajada_broca)"
        global bajar= pose_add ( get_actual_tcp_pose (), bajada_broca)
        $ 977 "bajar" "breakAfter"
        movel(bajar, a=0.005, v=0.001)
        $ 978 "subir≔pose_sub(get_actual_tcp_pose(), bajada_broca)"
        global subir= pose_sub ( get_actual_tcp_pose (), bajada_broca)
        $ 979 "subir" "breakAfter"
        movel(subir, a=0.01, v=0.01)
        $ 980 "bajada_broca≔pose_sub(bajada_broca, bajada)"
        global bajada_broca= pose_sub (bajada_broca, bajada)
        Loop_25 = Loop_25 + 1
      end
      $ 981 "Direction: Base Z+"
      global move_thread_flag_981=0
      thread move_thread_981():
        enter_critical
        move_thread_flag_981 = 1
        local towardsPos=calculate_point_to_move_towards(p[0.0,0.0,0.0,0.0,0.0,0.0], [0.0,0.0,1.0], 0.06)
        movel(towardsPos, a=0.035, v=0.03)
        move_thread_flag_981 = 2
        exit_critical
      end
      move_thread_flag_981 = 0
      move_thread_han_981 = run move_thread_981()
      while (True):
        sleep(1.0E-10)
        if (move_thread_flag_981 > 1):
          join move_thread_han_981
          $ 982 "Until (distance)"
          break
        end
        sync()
      end
      $ 983 "Set CO[1]=Apagar"
      set_configurable_digital_out(1, False)
      $ 984 "barreno_actual≔barreno_actual+1"
      global barreno_actual=barreno_actual+1
    end
    $ 987 "EF"
    $ 988 "'desbaste_inicial'"
    # 'desbaste_inicial'
    $ 989 "bajada_broca≔p[0,0,-0.012,0,0,0]"
    global bajada_broca=p[0,0,-0.012,0,0,0]
    $ 990 "barrenos_menos1≔8"
    global barrenos_menos1=8
    $ 991 "barreno_actual≔0"
    global barreno_actual=0
    $ 992 "Loop barreno_actual≤barrenos_menos1"
    while (barreno_actual <= barrenos_menos1):
      $ 993 "Perforacion"
      $ 994 "MoveL"
      $ 995 "internos≔interpolate_pose(Linea3_E, Linea3_F, barreno_actual/barrenos_menos1)"
      global internos= interpolate_pose (Linea3_E_p, Linea3_F_p, barreno_actual/barrenos_menos1)
      $ 996 "internos" "breakAfter"
      movel(internos, a=0.5, v=0.1)
      $ 997 "'desbaste_inicial'"
      # 'desbaste_inicial'
      $ 998 "bajada_broca≔p[0,0,-0.012,0,0,0]"
      global bajada_broca=p[0,0,-0.012,0,0,0]
      $ 999 "bajada≔p[0,0,0.012,0,0,0]"
      global bajada=p[0,0,0.012,0,0,0]
      $ 1000 "Direction: Base Z-"
      global move_thread_flag_1000=0
      thread move_thread_1000():
        enter_critical
        move_thread_flag_1000 = 1
        local towardsPos=calculate_point_to_move_towards(p[0.0,0.0,0.0,0.0,0.0,0.0], [0.0,0.0,-1.0], 0.055)
        movel(towardsPos, a=0.015, v=0.02)
        move_thread_flag_1000 = 2
        exit_critical
      end
      move_thread_flag_1000 = 0
      move_thread_han_1000 = run move_thread_1000()
      while (True):
        sleep(1.0E-10)
        if (move_thread_flag_1000 > 1):
          join move_thread_han_1000
          $ 1001 "Until (distance)"
          break
        end
        sync()
      end
      $ 1002 "Popup: punto contacto alanzdo"
      popup("punto contacto alanzdo", "Mensaje", False, False, blocking=True)
      $ 1003 "Direction: Base Z+"
      global move_thread_flag_1003=0
      thread move_thread_1003():
        enter_critical
        move_thread_flag_1003 = 1
        local towardsPos=calculate_point_to_move_towards(p[0.0,0.0,0.0,0.0,0.0,0.0], [0.0,0.0,1.0], 0.001)
        movel(towardsPos, a=0.005, v=0.003)
        move_thread_flag_1003 = 2
        exit_critical
      end
      move_thread_flag_1003 = 0
      move_thread_han_1003 = run move_thread_1003()
      while (True):
        sleep(1.0E-10)
        if (move_thread_flag_1003 > 1):
          join move_thread_han_1003
          $ 1004 "Until (distance)"
          break
        end
        sync()
      end
      $ 1005 "Wait: 0.3"
      sleep(0.3)
      $ 1006 "Set CO[1]=Encender"
      set_configurable_digital_out(1, True)
      $ 1007 "Wait: 0.3"
      sleep(0.3)
      $ 1008 "Loop 2 times"
      Loop_27 = 0
      while (Loop_27 < 2):
        $ 1009 "bajar≔pose_add(get_actual_tcp_pose(), bajada_broca)"
        global bajar= pose_add ( get_actual_tcp_pose (), bajada_broca)
        $ 1010 "bajar" "breakAfter"
        movel(bajar, a=0.005, v=0.001)
        $ 1011 "subir≔pose_sub(get_actual_tcp_pose(), bajada_broca)"
        global subir= pose_sub ( get_actual_tcp_pose (), bajada_broca)
        $ 1012 "subir" "breakAfter"
        movel(subir, a=0.01, v=0.01)
        $ 1013 "bajada_broca≔pose_sub(bajada_broca, bajada)"
        global bajada_broca= pose_sub (bajada_broca, bajada)
        Loop_27 = Loop_27 + 1
      end
      $ 1014 "Direction: Base Z+"
      global move_thread_flag_1014=0
      thread move_thread_1014():
        enter_critical
        move_thread_flag_1014 = 1
        local towardsPos=calculate_point_to_move_towards(p[0.0,0.0,0.0,0.0,0.0,0.0], [0.0,0.0,1.0], 0.06)
        movel(towardsPos, a=0.035, v=0.03)
        move_thread_flag_1014 = 2
        exit_critical
      end
      move_thread_flag_1014 = 0
      move_thread_han_1014 = run move_thread_1014()
      while (True):
        sleep(1.0E-10)
        if (move_thread_flag_1014 > 1):
          join move_thread_han_1014
          $ 1015 "Until (distance)"
          break
        end
        sync()
      end
      $ 1016 "Set CO[1]=Apagar"
      set_configurable_digital_out(1, False)
      $ 1017 "barreno_actual≔barreno_actual+1"
      global barreno_actual=barreno_actual+1
    end
    $ 1020 "Popup: Linea3 con media Terminada!"
    popup("Linea3 con media Terminada!", "Mensaje", False, False, blocking=True)
    $ 1021 "Linea4"
    $ 1022 "Marcar_puntos"
    $ 1023 "MoveL"
    $ 1024 "Home3" "breakAfter"
    movel(Home3_p, a=0.5, v=0.1)
    $ 1025 "Linea4_A" "breakAfter"
    movel(Linea4_A_p, a=0.5, v=0.1)
    $ 1026 "Linea4_B" "breakAfter"
    movel(Linea4_B_p, a=0.5, v=0.1)
    $ 1027 "Linea4_C" "breakAfter"
    movel(Linea4_C_p, a=0.5, v=0.1)
    $ 1028 "Linea4_D" "breakAfter"
    movel(Linea4_D_p, a=0.5, v=0.1)
    $ 1029 "Linea4_E" "breakAfter"
    movel(Linea4_E_p, a=0.5, v=0.1)
    $ 1030 "Linea4_F" "breakAfter"
    movel(Linea4_F_p, a=0.5, v=0.1)
    $ 1031 "AB"
    $ 1032 "'desbaste_inicial'"
    # 'desbaste_inicial'
    $ 1033 "bajada_broca≔p[0,0,-0.012,0,0,0]"
    global bajada_broca=p[0,0,-0.012,0,0,0]
    $ 1034 "barrenos_menos1≔8"
    global barrenos_menos1=8
    $ 1035 "barreno_actual≔0"
    global barreno_actual=0
    $ 1036 "Loop barreno_actual≤barrenos_menos1"
    while (barreno_actual <= barrenos_menos1):
      $ 1037 "Perforacion"
      $ 1038 "MoveL"
      $ 1039 "internos≔interpolate_pose(Linea4_A, Linea4_B, barreno_actual/barrenos_menos1)"
      global internos= interpolate_pose (Linea4_A_p, Linea4_B_p, barreno_actual/barrenos_menos1)
      $ 1040 "internos" "breakAfter"
      movel(internos, a=0.5, v=0.1)
      $ 1041 "'desbaste_inicial'"
      # 'desbaste_inicial'
      $ 1042 "bajada_broca≔p[0,0,-0.012,0,0,0]"
      global bajada_broca=p[0,0,-0.012,0,0,0]
      $ 1043 "bajada≔p[0,0,0.012,0,0,0]"
      global bajada=p[0,0,0.012,0,0,0]
      $ 1044 "Direction: Base Z-"
      global move_thread_flag_1044=0
      thread move_thread_1044():
        enter_critical
        move_thread_flag_1044 = 1
        local towardsPos=calculate_point_to_move_towards(p[0.0,0.0,0.0,0.0,0.0,0.0], [0.0,0.0,-1.0], 0.055)
        movel(towardsPos, a=0.015, v=0.02)
        move_thread_flag_1044 = 2
        exit_critical
      end
      move_thread_flag_1044 = 0
      move_thread_han_1044 = run move_thread_1044()
      while (True):
        sleep(1.0E-10)
        if (move_thread_flag_1044 > 1):
          join move_thread_han_1044
          $ 1045 "Until (distance)"
          break
        end
        sync()
      end
      $ 1046 "Popup: punto contacto alanzdo"
      popup("punto contacto alanzdo", "Mensaje", False, False, blocking=True)
      $ 1047 "Direction: Base Z+"
      global move_thread_flag_1047=0
      thread move_thread_1047():
        enter_critical
        move_thread_flag_1047 = 1
        local towardsPos=calculate_point_to_move_towards(p[0.0,0.0,0.0,0.0,0.0,0.0], [0.0,0.0,1.0], 0.001)
        movel(towardsPos, a=0.005, v=0.003)
        move_thread_flag_1047 = 2
        exit_critical
      end
      move_thread_flag_1047 = 0
      move_thread_han_1047 = run move_thread_1047()
      while (True):
        sleep(1.0E-10)
        if (move_thread_flag_1047 > 1):
          join move_thread_han_1047
          $ 1048 "Until (distance)"
          break
        end
        sync()
      end
      $ 1049 "Wait: 0.3"
      sleep(0.3)
      $ 1050 "Set CO[1]=Encender"
      set_configurable_digital_out(1, True)
      $ 1051 "Wait: 0.3"
      sleep(0.3)
      $ 1052 "Loop 2 times"
      Loop_29 = 0
      while (Loop_29 < 2):
        $ 1053 "bajar≔pose_add(get_actual_tcp_pose(), bajada_broca)"
        global bajar= pose_add ( get_actual_tcp_pose (), bajada_broca)
        $ 1054 "bajar" "breakAfter"
        movel(bajar, a=0.005, v=0.001)
        $ 1055 "subir≔pose_sub(get_actual_tcp_pose(), bajada_broca)"
        global subir= pose_sub ( get_actual_tcp_pose (), bajada_broca)
        $ 1056 "subir" "breakAfter"
        movel(subir, a=0.01, v=0.01)
        $ 1057 "bajada_broca≔pose_sub(bajada_broca, bajada)"
        global bajada_broca= pose_sub (bajada_broca, bajada)
        Loop_29 = Loop_29 + 1
      end
      $ 1058 "Direction: Base Z+"
      global move_thread_flag_1058=0
      thread move_thread_1058():
        enter_critical
        move_thread_flag_1058 = 1
        local towardsPos=calculate_point_to_move_towards(p[0.0,0.0,0.0,0.0,0.0,0.0], [0.0,0.0,1.0], 0.06)
        movel(towardsPos, a=0.035, v=0.03)
        move_thread_flag_1058 = 2
        exit_critical
      end
      move_thread_flag_1058 = 0
      move_thread_han_1058 = run move_thread_1058()
      while (True):
        sleep(1.0E-10)
        if (move_thread_flag_1058 > 1):
          join move_thread_han_1058
          $ 1059 "Until (distance)"
          break
        end
        sync()
      end
      $ 1060 "Set CO[1]=Apagar"
      set_configurable_digital_out(1, False)
      $ 1061 "barreno_actual≔barreno_actual+1"
      global barreno_actual=barreno_actual+1
    end
    $ 1064 "CD"
    $ 1065 "'desbaste_inicial'"
    # 'desbaste_inicial'
    $ 1066 "bajada_broca≔p[0,0,-0.012,0,0,0]"
    global bajada_broca=p[0,0,-0.012,0,0,0]
    $ 1067 "barrenos_menos1≔8"
    global barrenos_menos1=8
    $ 1068 "barreno_actual≔0"
    global barreno_actual=0
    $ 1069 "Loop barreno_actual≤barrenos_menos1"
    while (barreno_actual <= barrenos_menos1):
      $ 1070 "Perforacion"
      $ 1071 "MoveL"
      $ 1072 "internos≔interpolate_pose(Linea4_C, Linea4_D, barreno_actual/barrenos_menos1)"
      global internos= interpolate_pose (Linea4_C_p, Linea4_D_p, barreno_actual/barrenos_menos1)
      $ 1073 "internos" "breakAfter"
      movel(internos, a=0.5, v=0.1)
      $ 1074 "'desbaste_inicial'"
      # 'desbaste_inicial'
      $ 1075 "bajada_broca≔p[0,0,-0.012,0,0,0]"
      global bajada_broca=p[0,0,-0.012,0,0,0]
      $ 1076 "bajada≔p[0,0,0.012,0,0,0]"
      global bajada=p[0,0,0.012,0,0,0]
      $ 1077 "Direction: Base Z-"
      global move_thread_flag_1077=0
      thread move_thread_1077():
        enter_critical
        move_thread_flag_1077 = 1
        local towardsPos=calculate_point_to_move_towards(p[0.0,0.0,0.0,0.0,0.0,0.0], [0.0,0.0,-1.0], 0.055)
        movel(towardsPos, a=0.015, v=0.02)
        move_thread_flag_1077 = 2
        exit_critical
      end
      move_thread_flag_1077 = 0
      move_thread_han_1077 = run move_thread_1077()
      while (True):
        sleep(1.0E-10)
        if (move_thread_flag_1077 > 1):
          join move_thread_han_1077
          $ 1078 "Until (distance)"
          break
        end
        sync()
      end
      $ 1079 "Popup: punto contacto alanzdo"
      popup("punto contacto alanzdo", "Mensaje", False, False, blocking=True)
      $ 1080 "Direction: Base Z+"
      global move_thread_flag_1080=0
      thread move_thread_1080():
        enter_critical
        move_thread_flag_1080 = 1
        local towardsPos=calculate_point_to_move_towards(p[0.0,0.0,0.0,0.0,0.0,0.0], [0.0,0.0,1.0], 0.001)
        movel(towardsPos, a=0.005, v=0.003)
        move_thread_flag_1080 = 2
        exit_critical
      end
      move_thread_flag_1080 = 0
      move_thread_han_1080 = run move_thread_1080()
      while (True):
        sleep(1.0E-10)
        if (move_thread_flag_1080 > 1):
          join move_thread_han_1080
          $ 1081 "Until (distance)"
          break
        end
        sync()
      end
      $ 1082 "Wait: 0.3"
      sleep(0.3)
      $ 1083 "Set CO[1]=Encender"
      set_configurable_digital_out(1, True)
      $ 1084 "Wait: 0.3"
      sleep(0.3)
      $ 1085 "Loop 2 times"
      Loop_31 = 0
      while (Loop_31 < 2):
        $ 1086 "bajar≔pose_add(get_actual_tcp_pose(), bajada_broca)"
        global bajar= pose_add ( get_actual_tcp_pose (), bajada_broca)
        $ 1087 "bajar" "breakAfter"
        movel(bajar, a=0.005, v=0.001)
        $ 1088 "subir≔pose_sub(get_actual_tcp_pose(), bajada_broca)"
        global subir= pose_sub ( get_actual_tcp_pose (), bajada_broca)
        $ 1089 "subir" "breakAfter"
        movel(subir, a=0.01, v=0.01)
        $ 1090 "bajada_broca≔pose_sub(bajada_broca, bajada)"
        global bajada_broca= pose_sub (bajada_broca, bajada)
        Loop_31 = Loop_31 + 1
      end
      $ 1091 "Direction: Base Z+"
      global move_thread_flag_1091=0
      thread move_thread_1091():
        enter_critical
        move_thread_flag_1091 = 1
        local towardsPos=calculate_point_to_move_towards(p[0.0,0.0,0.0,0.0,0.0,0.0], [0.0,0.0,1.0], 0.06)
        movel(towardsPos, a=0.035, v=0.03)
        move_thread_flag_1091 = 2
        exit_critical
      end
      move_thread_flag_1091 = 0
      move_thread_han_1091 = run move_thread_1091()
      while (True):
        sleep(1.0E-10)
        if (move_thread_flag_1091 > 1):
          join move_thread_han_1091
          $ 1092 "Until (distance)"
          break
        end
        sync()
      end
      $ 1093 "Set CO[1]=Apagar"
      set_configurable_digital_out(1, False)
      $ 1094 "barreno_actual≔barreno_actual+1"
      global barreno_actual=barreno_actual+1
    end
    $ 1097 "EF"
    $ 1098 "'desbaste_inicial'"
    # 'desbaste_inicial'
    $ 1099 "bajada_broca≔p[0,0,-0.012,0,0,0]"
    global bajada_broca=p[0,0,-0.012,0,0,0]
    $ 1100 "barrenos_menos1≔8"
    global barrenos_menos1=8
    $ 1101 "barreno_actual≔0"
    global barreno_actual=0
    $ 1102 "Loop barreno_actual≤barrenos_menos1"
    while (barreno_actual <= barrenos_menos1):
      $ 1103 "Perforacion"
      $ 1104 "MoveL"
      $ 1105 "internos≔interpolate_pose(Linea4_E, Linea4_F, barreno_actual/barrenos_menos1)"
      global internos= interpolate_pose (Linea4_E_p, Linea4_F_p, barreno_actual/barrenos_menos1)
      $ 1106 "internos" "breakAfter"
      movel(internos, a=0.5, v=0.1)
      $ 1107 "'desbaste_inicial'"
      # 'desbaste_inicial'
      $ 1108 "bajada_broca≔p[0,0,-0.012,0,0,0]"
      global bajada_broca=p[0,0,-0.012,0,0,0]
      $ 1109 "bajada≔p[0,0,0.012,0,0,0]"
      global bajada=p[0,0,0.012,0,0,0]
      $ 1110 "Direction: Base Z-"
      global move_thread_flag_1110=0
      thread move_thread_1110():
        enter_critical
        move_thread_flag_1110 = 1
        local towardsPos=calculate_point_to_move_towards(p[0.0,0.0,0.0,0.0,0.0,0.0], [0.0,0.0,-1.0], 0.055)
        movel(towardsPos, a=0.015, v=0.02)
        move_thread_flag_1110 = 2
        exit_critical
      end
      move_thread_flag_1110 = 0
      move_thread_han_1110 = run move_thread_1110()
      while (True):
        sleep(1.0E-10)
        if (move_thread_flag_1110 > 1):
          join move_thread_han_1110
          $ 1111 "Until (distance)"
          break
        end
        sync()
      end
      $ 1112 "Popup: punto contacto alanzdo"
      popup("punto contacto alanzdo", "Mensaje", False, False, blocking=True)
      $ 1113 "Direction: Base Z+"
      global move_thread_flag_1113=0
      thread move_thread_1113():
        enter_critical
        move_thread_flag_1113 = 1
        local towardsPos=calculate_point_to_move_towards(p[0.0,0.0,0.0,0.0,0.0,0.0], [0.0,0.0,1.0], 0.001)
        movel(towardsPos, a=0.005, v=0.003)
        move_thread_flag_1113 = 2
        exit_critical
      end
      move_thread_flag_1113 = 0
      move_thread_han_1113 = run move_thread_1113()
      while (True):
        sleep(1.0E-10)
        if (move_thread_flag_1113 > 1):
          join move_thread_han_1113
          $ 1114 "Until (distance)"
          break
        end
        sync()
      end
      $ 1115 "Wait: 0.3"
      sleep(0.3)
      $ 1116 "Set CO[1]=Encender"
      set_configurable_digital_out(1, True)
      $ 1117 "Wait: 0.3"
      sleep(0.3)
      $ 1118 "Loop 2 times"
      Loop_33 = 0
      while (Loop_33 < 2):
        $ 1119 "bajar≔pose_add(get_actual_tcp_pose(), bajada_broca)"
        global bajar= pose_add ( get_actual_tcp_pose (), bajada_broca)
        $ 1120 "bajar" "breakAfter"
        movel(bajar, a=0.005, v=0.001)
        $ 1121 "subir≔pose_sub(get_actual_tcp_pose(), bajada_broca)"
        global subir= pose_sub ( get_actual_tcp_pose (), bajada_broca)
        $ 1122 "subir" "breakAfter"
        movel(subir, a=0.01, v=0.01)
        $ 1123 "bajada_broca≔pose_sub(bajada_broca, bajada)"
        global bajada_broca= pose_sub (bajada_broca, bajada)
        Loop_33 = Loop_33 + 1
      end
      $ 1124 "Direction: Base Z+"
      global move_thread_flag_1124=0
      thread move_thread_1124():
        enter_critical
        move_thread_flag_1124 = 1
        local towardsPos=calculate_point_to_move_towards(p[0.0,0.0,0.0,0.0,0.0,0.0], [0.0,0.0,1.0], 0.06)
        movel(towardsPos, a=0.035, v=0.03)
        move_thread_flag_1124 = 2
        exit_critical
      end
      move_thread_flag_1124 = 0
      move_thread_han_1124 = run move_thread_1124()
      while (True):
        sleep(1.0E-10)
        if (move_thread_flag_1124 > 1):
          join move_thread_han_1124
          $ 1125 "Until (distance)"
          break
        end
        sync()
      end
      $ 1126 "Set CO[1]=Apagar"
      set_configurable_digital_out(1, False)
      $ 1127 "barreno_actual≔barreno_actual+1"
      global barreno_actual=barreno_actual+1
      $ 1128 "If barreno_actual≥barrenos_menos1"
      if (barreno_actual >= barrenos_menos1):
        $ 1129 "cambiar_broca≔ True "
        global cambiar_broca=  True
      end
    end
    $ 1132 "Popup: Linea4 con media Terminada!"
    popup("Linea4 con media Terminada!", "Mensaje", False, False, blocking=True)
    $ 1133 "Broca_3"
    $ 1134 "Linea3"
    $ 1135 "Marcar_puntos"
    $ 1136 "MoveL"
    $ 1137 "Home3" "breakAfter"
    movel(Home3_p, a=0.5, v=0.1)
    $ 1138 "Linea3_A" "breakAfter"
    movel(Linea3_A_p, a=0.5, v=0.1)
    $ 1139 "Linea3_B" "breakAfter"
    movel(Linea3_B_p, a=0.5, v=0.1)
    $ 1140 "Linea3_C" "breakAfter"
    movel(Linea3_C_p, a=0.5, v=0.1)
    $ 1141 "Linea3_D" "breakAfter"
    movel(Linea3_D_p, a=0.5, v=0.1)
    $ 1142 "Linea3_E" "breakAfter"
    movel(Linea3_E_p, a=0.5, v=0.1)
    $ 1143 "Linea3_F" "breakAfter"
    movel(Linea3_F_p, a=0.5, v=0.1)
    $ 1144 "AB"
    $ 1145 "'desbaste_inicial'"
    # 'desbaste_inicial'
    $ 1146 "bajada_broca≔p[0,0,-0.024,0,0,0]"
    global bajada_broca=p[0,0,-0.024,0,0,0]
    $ 1147 "barrenos_menos1≔8"
    global barrenos_menos1=8
    $ 1148 "barreno_actual≔0"
    global barreno_actual=0
    $ 1149 "Loop barreno_actual≤barrenos_menos1"
    while (barreno_actual <= barrenos_menos1):
      $ 1150 "Perforacion"
      $ 1151 "MoveL"
      $ 1152 "internos≔interpolate_pose(Linea3_A, Linea3_B, barreno_actual/barrenos_menos1)"
      global internos= interpolate_pose (Linea3_A_p, Linea3_B_p, barreno_actual/barrenos_menos1)
      $ 1153 "internos" "breakAfter"
      movel(internos, a=0.5, v=0.1)
      $ 1154 "'desbaste_inicial'"
      # 'desbaste_inicial'
      $ 1155 "bajada_broca≔p[0,0,-0.024,0,0,0]"
      global bajada_broca=p[0,0,-0.024,0,0,0]
      $ 1156 "bajada≔p[0,0,0.024,0,0,0]"
      global bajada=p[0,0,0.024,0,0,0]
      $ 1157 "Direction: Base Z-"
      global move_thread_flag_1157=0
      thread move_thread_1157():
        enter_critical
        move_thread_flag_1157 = 1
        local towardsPos=calculate_point_to_move_towards(p[0.0,0.0,0.0,0.0,0.0,0.0], [0.0,0.0,-1.0], 0.055)
        movel(towardsPos, a=0.015, v=0.02)
        move_thread_flag_1157 = 2
        exit_critical
      end
      move_thread_flag_1157 = 0
      move_thread_han_1157 = run move_thread_1157()
      while (True):
        sleep(1.0E-10)
        if (move_thread_flag_1157 > 1):
          join move_thread_han_1157
          $ 1158 "Until (distance)"
          break
        end
        sync()
      end
      $ 1159 "Popup: punto contacto alanzdo"
      popup("punto contacto alanzdo", "Mensaje", False, False, blocking=True)
      $ 1160 "Direction: Base Z+"
      global move_thread_flag_1160=0
      thread move_thread_1160():
        enter_critical
        move_thread_flag_1160 = 1
        local towardsPos=calculate_point_to_move_towards(p[0.0,0.0,0.0,0.0,0.0,0.0], [0.0,0.0,1.0], 0.001)
        movel(towardsPos, a=0.005, v=0.003)
        move_thread_flag_1160 = 2
        exit_critical
      end
      move_thread_flag_1160 = 0
      move_thread_han_1160 = run move_thread_1160()
      while (True):
        sleep(1.0E-10)
        if (move_thread_flag_1160 > 1):
          join move_thread_han_1160
          $ 1161 "Until (distance)"
          break
        end
        sync()
      end
      $ 1162 "Wait: 0.3"
      sleep(0.3)
      $ 1163 "Set CO[1]=Encender"
      set_configurable_digital_out(1, True)
      $ 1164 "Wait: 0.3"
      sleep(0.3)
      $ 1165 "Loop 1 times"
      Loop_37 = 0
      while (Loop_37 < 1):
        $ 1166 "bajar≔pose_add(get_actual_tcp_pose(), bajada_broca)"
        global bajar= pose_add ( get_actual_tcp_pose (), bajada_broca)
        $ 1167 "bajar" "breakAfter"
        movel(bajar, a=0.005, v=0.001)
        $ 1168 "subir≔pose_sub(get_actual_tcp_pose(), bajada_broca)"
        global subir= pose_sub ( get_actual_tcp_pose (), bajada_broca)
        $ 1169 "subir" "breakAfter"
        movel(subir, a=0.01, v=0.01)
        $ 1170 "bajada_broca≔pose_sub(bajada_broca, bajada)"
        global bajada_broca= pose_sub (bajada_broca, bajada)
        Loop_37 = Loop_37 + 1
      end
      $ 1171 "Direction: Base Z+"
      global move_thread_flag_1171=0
      thread move_thread_1171():
        enter_critical
        move_thread_flag_1171 = 1
        local towardsPos=calculate_point_to_move_towards(p[0.0,0.0,0.0,0.0,0.0,0.0], [0.0,0.0,1.0], 0.06)
        movel(towardsPos, a=0.035, v=0.03)
        move_thread_flag_1171 = 2
        exit_critical
      end
      move_thread_flag_1171 = 0
      move_thread_han_1171 = run move_thread_1171()
      while (True):
        sleep(1.0E-10)
        if (move_thread_flag_1171 > 1):
          join move_thread_han_1171
          $ 1172 "Until (distance)"
          break
        end
        sync()
      end
      $ 1173 "Set CO[1]=Apagar"
      set_configurable_digital_out(1, False)
      $ 1174 "barreno_actual≔barreno_actual+1"
      global barreno_actual=barreno_actual+1
    end
    $ 1177 "CD"
    $ 1178 "'desbaste_inicial'"
    # 'desbaste_inicial'
    $ 1179 "bajada_broca≔p[0,0,-0.024,0,0,0]"
    global bajada_broca=p[0,0,-0.024,0,0,0]
    $ 1180 "barrenos_menos1≔8"
    global barrenos_menos1=8
    $ 1181 "barreno_actual≔0"
    global barreno_actual=0
    $ 1182 "Loop barreno_actual≤barrenos_menos1"
    while (barreno_actual <= barrenos_menos1):
      $ 1183 "Perforacion"
      $ 1184 "MoveL"
      $ 1185 "internos≔interpolate_pose(Linea3_C, Linea3_D, barreno_actual/barrenos_menos1)"
      global internos= interpolate_pose (Linea3_C_p, Linea3_D_p, barreno_actual/barrenos_menos1)
      $ 1186 "internos" "breakAfter"
      movel(internos, a=0.5, v=0.1)
      $ 1187 "'desbaste_inicial'"
      # 'desbaste_inicial'
      $ 1188 "bajada_broca≔p[0,0,-0.024,0,0,0]"
      global bajada_broca=p[0,0,-0.024,0,0,0]
      $ 1189 "bajada≔p[0,0,0.024,0,0,0]"
      global bajada=p[0,0,0.024,0,0,0]
      $ 1190 "Direction: Base Z-"
      global move_thread_flag_1190=0
      thread move_thread_1190():
        enter_critical
        move_thread_flag_1190 = 1
        local towardsPos=calculate_point_to_move_towards(p[0.0,0.0,0.0,0.0,0.0,0.0], [0.0,0.0,-1.0], 0.055)
        movel(towardsPos, a=0.015, v=0.02)
        move_thread_flag_1190 = 2
        exit_critical
      end
      move_thread_flag_1190 = 0
      move_thread_han_1190 = run move_thread_1190()
      while (True):
        sleep(1.0E-10)
        if (move_thread_flag_1190 > 1):
          join move_thread_han_1190
          $ 1191 "Until (distance)"
          break
        end
        sync()
      end
      $ 1192 "Popup: punto contacto alanzdo"
      popup("punto contacto alanzdo", "Mensaje", False, False, blocking=True)
      $ 1193 "Direction: Base Z+"
      global move_thread_flag_1193=0
      thread move_thread_1193():
        enter_critical
        move_thread_flag_1193 = 1
        local towardsPos=calculate_point_to_move_towards(p[0.0,0.0,0.0,0.0,0.0,0.0], [0.0,0.0,1.0], 0.001)
        movel(towardsPos, a=0.005, v=0.003)
        move_thread_flag_1193 = 2
        exit_critical
      end
      move_thread_flag_1193 = 0
      move_thread_han_1193 = run move_thread_1193()
      while (True):
        sleep(1.0E-10)
        if (move_thread_flag_1193 > 1):
          join move_thread_han_1193
          $ 1194 "Until (distance)"
          break
        end
        sync()
      end
      $ 1195 "Wait: 0.3"
      sleep(0.3)
      $ 1196 "Set CO[1]=Encender"
      set_configurable_digital_out(1, True)
      $ 1197 "Wait: 0.3"
      sleep(0.3)
      $ 1198 "Loop 1 times"
      Loop_41 = 0
      while (Loop_41 < 1):
        $ 1199 "bajar≔pose_add(get_actual_tcp_pose(), bajada_broca)"
        global bajar= pose_add ( get_actual_tcp_pose (), bajada_broca)
        $ 1200 "bajar" "breakAfter"
        movel(bajar, a=0.005, v=0.001)
        $ 1201 "subir≔pose_sub(get_actual_tcp_pose(), bajada_broca)"
        global subir= pose_sub ( get_actual_tcp_pose (), bajada_broca)
        $ 1202 "subir" "breakAfter"
        movel(subir, a=0.01, v=0.01)
        $ 1203 "bajada_broca≔pose_sub(bajada_broca, bajada)"
        global bajada_broca= pose_sub (bajada_broca, bajada)
        Loop_41 = Loop_41 + 1
      end
      $ 1204 "Direction: Base Z+"
      global move_thread_flag_1204=0
      thread move_thread_1204():
        enter_critical
        move_thread_flag_1204 = 1
        local towardsPos=calculate_point_to_move_towards(p[0.0,0.0,0.0,0.0,0.0,0.0], [0.0,0.0,1.0], 0.06)
        movel(towardsPos, a=0.035, v=0.03)
        move_thread_flag_1204 = 2
        exit_critical
      end
      move_thread_flag_1204 = 0
      move_thread_han_1204 = run move_thread_1204()
      while (True):
        sleep(1.0E-10)
        if (move_thread_flag_1204 > 1):
          join move_thread_han_1204
          $ 1205 "Until (distance)"
          break
        end
        sync()
      end
      $ 1206 "Set CO[1]=Apagar"
      set_configurable_digital_out(1, False)
      $ 1207 "barreno_actual≔barreno_actual+1"
      global barreno_actual=barreno_actual+1
    end
    $ 1210 "EF"
    $ 1211 "'desbaste_inicial'"
    # 'desbaste_inicial'
    $ 1212 "bajada_broca≔p[0,0,-0.024,0,0,0]"
    global bajada_broca=p[0,0,-0.024,0,0,0]
    $ 1213 "barrenos_menos1≔8"
    global barrenos_menos1=8
    $ 1214 "barreno_actual≔0"
    global barreno_actual=0
    $ 1215 "Loop barreno_actual≤barrenos_menos1"
    while (barreno_actual <= barrenos_menos1):
      $ 1216 "Perforacion"
      $ 1217 "MoveL"
      $ 1218 "internos≔interpolate_pose(Linea3_E, Linea3_F, barreno_actual/barrenos_menos1)"
      global internos= interpolate_pose (Linea3_E_p, Linea3_F_p, barreno_actual/barrenos_menos1)
      $ 1219 "internos" "breakAfter"
      movel(internos, a=0.5, v=0.1)
      $ 1220 "'desbaste_inicial'"
      # 'desbaste_inicial'
      $ 1221 "bajada_broca≔p[0,0,-0.024,0,0,0]"
      global bajada_broca=p[0,0,-0.024,0,0,0]
      $ 1222 "bajada≔p[0,0,0.024,0,0,0]"
      global bajada=p[0,0,0.024,0,0,0]
      $ 1223 "Direction: Base Z-"
      global move_thread_flag_1223=0
      thread move_thread_1223():
        enter_critical
        move_thread_flag_1223 = 1
        local towardsPos=calculate_point_to_move_towards(p[0.0,0.0,0.0,0.0,0.0,0.0], [0.0,0.0,-1.0], 0.055)
        movel(towardsPos, a=0.015, v=0.02)
        move_thread_flag_1223 = 2
        exit_critical
      end
      move_thread_flag_1223 = 0
      move_thread_han_1223 = run move_thread_1223()
      while (True):
        sleep(1.0E-10)
        if (move_thread_flag_1223 > 1):
          join move_thread_han_1223
          $ 1224 "Until (distance)"
          break
        end
        sync()
      end
      $ 1225 "Popup: punto contacto alanzdo"
      popup("punto contacto alanzdo", "Mensaje", False, False, blocking=True)
      $ 1226 "Direction: Base Z+"
      global move_thread_flag_1226=0
      thread move_thread_1226():
        enter_critical
        move_thread_flag_1226 = 1
        local towardsPos=calculate_point_to_move_towards(p[0.0,0.0,0.0,0.0,0.0,0.0], [0.0,0.0,1.0], 0.001)
        movel(towardsPos, a=0.005, v=0.003)
        move_thread_flag_1226 = 2
        exit_critical
      end
      move_thread_flag_1226 = 0
      move_thread_han_1226 = run move_thread_1226()
      while (True):
        sleep(1.0E-10)
        if (move_thread_flag_1226 > 1):
          join move_thread_han_1226
          $ 1227 "Until (distance)"
          break
        end
        sync()
      end
      $ 1228 "Wait: 0.3"
      sleep(0.3)
      $ 1229 "Set CO[1]=Encender"
      set_configurable_digital_out(1, True)
      $ 1230 "Wait: 0.3"
      sleep(0.3)
      $ 1231 "Loop 1 times"
      Loop_45 = 0
      while (Loop_45 < 1):
        $ 1232 "bajar≔pose_add(get_actual_tcp_pose(), bajada_broca)"
        global bajar= pose_add ( get_actual_tcp_pose (), bajada_broca)
        $ 1233 "bajar" "breakAfter"
        movel(bajar, a=0.005, v=0.001)
        $ 1234 "subir≔pose_sub(get_actual_tcp_pose(), bajada_broca)"
        global subir= pose_sub ( get_actual_tcp_pose (), bajada_broca)
        $ 1235 "subir" "breakAfter"
        movel(subir, a=0.01, v=0.01)
        $ 1236 "bajada_broca≔pose_sub(bajada_broca, bajada)"
        global bajada_broca= pose_sub (bajada_broca, bajada)
        Loop_45 = Loop_45 + 1
      end
      $ 1237 "Direction: Base Z+"
      global move_thread_flag_1237=0
      thread move_thread_1237():
        enter_critical
        move_thread_flag_1237 = 1
        local towardsPos=calculate_point_to_move_towards(p[0.0,0.0,0.0,0.0,0.0,0.0], [0.0,0.0,1.0], 0.06)
        movel(towardsPos, a=0.035, v=0.03)
        move_thread_flag_1237 = 2
        exit_critical
      end
      move_thread_flag_1237 = 0
      move_thread_han_1237 = run move_thread_1237()
      while (True):
        sleep(1.0E-10)
        if (move_thread_flag_1237 > 1):
          join move_thread_han_1237
          $ 1238 "Until (distance)"
          break
        end
        sync()
      end
      $ 1239 "Set CO[1]=Apagar"
      set_configurable_digital_out(1, False)
      $ 1240 "barreno_actual≔barreno_actual+1"
      global barreno_actual=barreno_actual+1
    end
    $ 1243 "Popup: Linea3 con full Terminada!"
    popup("Linea3 con full Terminada!", "Mensaje", False, False, blocking=True)
    $ 1244 "Linea4"
    $ 1245 "Marcar_puntos"
    $ 1246 "MoveL"
    $ 1247 "Home3" "breakAfter"
    movel(Home3_p, a=0.5, v=0.1)
    $ 1248 "Linea4_A" "breakAfter"
    movel(Linea4_A_p, a=0.5, v=0.1)
    $ 1249 "Linea4_B" "breakAfter"
    movel(Linea4_B_p, a=0.5, v=0.1)
    $ 1250 "Linea4_C" "breakAfter"
    movel(Linea4_C_p, a=0.5, v=0.1)
    $ 1251 "Linea4_D" "breakAfter"
    movel(Linea4_D_p, a=0.5, v=0.1)
    $ 1252 "Linea4_E" "breakAfter"
    movel(Linea4_E_p, a=0.5, v=0.1)
    $ 1253 "Linea4_F" "breakAfter"
    movel(Linea4_F_p, a=0.5, v=0.1)
    $ 1254 "AB"
    $ 1255 "'desbaste_inicial'"
    # 'desbaste_inicial'
    $ 1256 "bajada_broca≔p[0,0,-0.024,0,0,0]"
    global bajada_broca=p[0,0,-0.024,0,0,0]
    $ 1257 "barrenos_menos1≔8"
    global barrenos_menos1=8
    $ 1258 "barreno_actual≔0"
    global barreno_actual=0
    $ 1259 "Loop barreno_actual≤barrenos_menos1"
    while (barreno_actual <= barrenos_menos1):
      $ 1260 "Perforacion"
      $ 1261 "MoveL"
      $ 1262 "internos≔interpolate_pose(Linea4_A, Linea4_B, barreno_actual/barrenos_menos1)"
      global internos= interpolate_pose (Linea4_A_p, Linea4_B_p, barreno_actual/barrenos_menos1)
      $ 1263 "internos" "breakAfter"
      movel(internos, a=0.5, v=0.1)
      $ 1264 "'desbaste_inicial'"
      # 'desbaste_inicial'
      $ 1265 "bajada_broca≔p[0,0,-0.024,0,0,0]"
      global bajada_broca=p[0,0,-0.024,0,0,0]
      $ 1266 "bajada≔p[0,0,0.024,0,0,0]"
      global bajada=p[0,0,0.024,0,0,0]
      $ 1267 "Direction: Base Z-"
      global move_thread_flag_1267=0
      thread move_thread_1267():
        enter_critical
        move_thread_flag_1267 = 1
        local towardsPos=calculate_point_to_move_towards(p[0.0,0.0,0.0,0.0,0.0,0.0], [0.0,0.0,-1.0], 0.055)
        movel(towardsPos, a=0.015, v=0.02)
        move_thread_flag_1267 = 2
        exit_critical
      end
      move_thread_flag_1267 = 0
      move_thread_han_1267 = run move_thread_1267()
      while (True):
        sleep(1.0E-10)
        if (move_thread_flag_1267 > 1):
          join move_thread_han_1267
          $ 1268 "Until (distance)"
          break
        end
        sync()
      end
      $ 1269 "Popup: punto contacto alanzdo"
      popup("punto contacto alanzdo", "Mensaje", False, False, blocking=True)
      $ 1270 "Direction: Base Z+"
      global move_thread_flag_1270=0
      thread move_thread_1270():
        enter_critical
        move_thread_flag_1270 = 1
        local towardsPos=calculate_point_to_move_towards(p[0.0,0.0,0.0,0.0,0.0,0.0], [0.0,0.0,1.0], 0.001)
        movel(towardsPos, a=0.005, v=0.003)
        move_thread_flag_1270 = 2
        exit_critical
      end
      move_thread_flag_1270 = 0
      move_thread_han_1270 = run move_thread_1270()
      while (True):
        sleep(1.0E-10)
        if (move_thread_flag_1270 > 1):
          join move_thread_han_1270
          $ 1271 "Until (distance)"
          break
        end
        sync()
      end
      $ 1272 "Wait: 0.3"
      sleep(0.3)
      $ 1273 "Set CO[1]=Encender"
      set_configurable_digital_out(1, True)
      $ 1274 "Wait: 0.3"
      sleep(0.3)
      $ 1275 "Loop 1 times"
      Loop_49 = 0
      while (Loop_49 < 1):
        $ 1276 "bajar≔pose_add(get_actual_tcp_pose(), bajada_broca)"
        global bajar= pose_add ( get_actual_tcp_pose (), bajada_broca)
        $ 1277 "bajar" "breakAfter"
        movel(bajar, a=0.005, v=0.001)
        $ 1278 "subir≔pose_sub(get_actual_tcp_pose(), bajada_broca)"
        global subir= pose_sub ( get_actual_tcp_pose (), bajada_broca)
        $ 1279 "subir" "breakAfter"
        movel(subir, a=0.01, v=0.01)
        $ 1280 "bajada_broca≔pose_sub(bajada_broca, bajada)"
        global bajada_broca= pose_sub (bajada_broca, bajada)
        Loop_49 = Loop_49 + 1
      end
      $ 1281 "Direction: Base Z+"
      global move_thread_flag_1281=0
      thread move_thread_1281():
        enter_critical
        move_thread_flag_1281 = 1
        local towardsPos=calculate_point_to_move_towards(p[0.0,0.0,0.0,0.0,0.0,0.0], [0.0,0.0,1.0], 0.06)
        movel(towardsPos, a=0.035, v=0.03)
        move_thread_flag_1281 = 2
        exit_critical
      end
      move_thread_flag_1281 = 0
      move_thread_han_1281 = run move_thread_1281()
      while (True):
        sleep(1.0E-10)
        if (move_thread_flag_1281 > 1):
          join move_thread_han_1281
          $ 1282 "Until (distance)"
          break
        end
        sync()
      end
      $ 1283 "Set CO[1]=Apagar"
      set_configurable_digital_out(1, False)
      $ 1284 "barreno_actual≔barreno_actual+1"
      global barreno_actual=barreno_actual+1
    end
    $ 1287 "CD"
    $ 1288 "'desbaste_inicial'"
    # 'desbaste_inicial'
    $ 1289 "bajada_broca≔p[0,0,-0.024,0,0,0]"
    global bajada_broca=p[0,0,-0.024,0,0,0]
    $ 1290 "barrenos_menos1≔8"
    global barrenos_menos1=8
    $ 1291 "barreno_actual≔0"
    global barreno_actual=0
    $ 1292 "Loop barreno_actual≤barrenos_menos1"
    while (barreno_actual <= barrenos_menos1):
      $ 1293 "Perforacion"
      $ 1294 "MoveL"
      $ 1295 "internos≔interpolate_pose(Linea4_C, Linea4_D, barreno_actual/barrenos_menos1)"
      global internos= interpolate_pose (Linea4_C_p, Linea4_D_p, barreno_actual/barrenos_menos1)
      $ 1296 "internos" "breakAfter"
      movel(internos, a=0.5, v=0.1)
      $ 1297 "'desbaste_inicial'"
      # 'desbaste_inicial'
      $ 1298 "bajada_broca≔p[0,0,-0.024,0,0,0]"
      global bajada_broca=p[0,0,-0.024,0,0,0]
      $ 1299 "bajada≔p[0,0,0.024,0,0,0]"
      global bajada=p[0,0,0.024,0,0,0]
      $ 1300 "Direction: Base Z-"
      global move_thread_flag_1300=0
      thread move_thread_1300():
        enter_critical
        move_thread_flag_1300 = 1
        local towardsPos=calculate_point_to_move_towards(p[0.0,0.0,0.0,0.0,0.0,0.0], [0.0,0.0,-1.0], 0.055)
        movel(towardsPos, a=0.015, v=0.02)
        move_thread_flag_1300 = 2
        exit_critical
      end
      move_thread_flag_1300 = 0
      move_thread_han_1300 = run move_thread_1300()
      while (True):
        sleep(1.0E-10)
        if (move_thread_flag_1300 > 1):
          join move_thread_han_1300
          $ 1301 "Until (distance)"
          break
        end
        sync()
      end
      $ 1302 "Popup: punto contacto alanzdo"
      popup("punto contacto alanzdo", "Mensaje", False, False, blocking=True)
      $ 1303 "Direction: Base Z+"
      global move_thread_flag_1303=0
      thread move_thread_1303():
        enter_critical
        move_thread_flag_1303 = 1
        local towardsPos=calculate_point_to_move_towards(p[0.0,0.0,0.0,0.0,0.0,0.0], [0.0,0.0,1.0], 0.001)
        movel(towardsPos, a=0.005, v=0.003)
        move_thread_flag_1303 = 2
        exit_critical
      end
      move_thread_flag_1303 = 0
      move_thread_han_1303 = run move_thread_1303()
      while (True):
        sleep(1.0E-10)
        if (move_thread_flag_1303 > 1):
          join move_thread_han_1303
          $ 1304 "Until (distance)"
          break
        end
        sync()
      end
      $ 1305 "Wait: 0.3"
      sleep(0.3)
      $ 1306 "Set CO[1]=Encender"
      set_configurable_digital_out(1, True)
      $ 1307 "Wait: 0.3"
      sleep(0.3)
      $ 1308 "Loop 1 times"
      Loop_52 = 0
      while (Loop_52 < 1):
        $ 1309 "bajar≔pose_add(get_actual_tcp_pose(), bajada_broca)"
        global bajar= pose_add ( get_actual_tcp_pose (), bajada_broca)
        $ 1310 "bajar" "breakAfter"
        movel(bajar, a=0.005, v=0.001)
        $ 1311 "subir≔pose_sub(get_actual_tcp_pose(), bajada_broca)"
        global subir= pose_sub ( get_actual_tcp_pose (), bajada_broca)
        $ 1312 "subir" "breakAfter"
        movel(subir, a=0.01, v=0.01)
        $ 1313 "bajada_broca≔pose_sub(bajada_broca, bajada)"
        global bajada_broca= pose_sub (bajada_broca, bajada)
        Loop_52 = Loop_52 + 1
      end
      $ 1314 "Direction: Base Z+"
      global move_thread_flag_1314=0
      thread move_thread_1314():
        enter_critical
        move_thread_flag_1314 = 1
        local towardsPos=calculate_point_to_move_towards(p[0.0,0.0,0.0,0.0,0.0,0.0], [0.0,0.0,1.0], 0.06)
        movel(towardsPos, a=0.035, v=0.03)
        move_thread_flag_1314 = 2
        exit_critical
      end
      move_thread_flag_1314 = 0
      move_thread_han_1314 = run move_thread_1314()
      while (True):
        sleep(1.0E-10)
        if (move_thread_flag_1314 > 1):
          join move_thread_han_1314
          $ 1315 "Until (distance)"
          break
        end
        sync()
      end
      $ 1316 "Set CO[1]=Apagar"
      set_configurable_digital_out(1, False)
      $ 1317 "barreno_actual≔barreno_actual+1"
      global barreno_actual=barreno_actual+1
    end
    $ 1320 "EF"
    $ 1321 "'desbaste_inicial'"
    # 'desbaste_inicial'
    $ 1322 "bajada_broca≔p[0,0,-0.024,0,0,0]"
    global bajada_broca=p[0,0,-0.024,0,0,0]
    $ 1323 "barrenos_menos1≔8"
    global barrenos_menos1=8
    $ 1324 "barreno_actual≔0"
    global barreno_actual=0
    $ 1325 "Loop barreno_actual≤barrenos_menos1"
    while (barreno_actual <= barrenos_menos1):
      $ 1326 "Perforacion"
      $ 1327 "MoveL"
      $ 1328 "internos≔interpolate_pose(Linea4_E, Linea4_F, barreno_actual/barrenos_menos1)"
      global internos= interpolate_pose (Linea4_E_p, Linea4_F_p, barreno_actual/barrenos_menos1)
      $ 1329 "internos" "breakAfter"
      movel(internos, a=0.5, v=0.1)
      $ 1330 "'desbaste_inicial'"
      # 'desbaste_inicial'
      $ 1331 "bajada_broca≔p[0,0,-0.024,0,0,0]"
      global bajada_broca=p[0,0,-0.024,0,0,0]
      $ 1332 "bajada≔p[0,0,0.024,0,0,0]"
      global bajada=p[0,0,0.024,0,0,0]
      $ 1333 "Direction: Base Z-"
      global move_thread_flag_1333=0
      thread move_thread_1333():
        enter_critical
        move_thread_flag_1333 = 1
        local towardsPos=calculate_point_to_move_towards(p[0.0,0.0,0.0,0.0,0.0,0.0], [0.0,0.0,-1.0], 0.055)
        movel(towardsPos, a=0.015, v=0.02)
        move_thread_flag_1333 = 2
        exit_critical
      end
      move_thread_flag_1333 = 0
      move_thread_han_1333 = run move_thread_1333()
      while (True):
        sleep(1.0E-10)
        if (move_thread_flag_1333 > 1):
          join move_thread_han_1333
          $ 1334 "Until (distance)"
          break
        end
        sync()
      end
      $ 1335 "Popup: punto contacto alanzdo"
      popup("punto contacto alanzdo", "Mensaje", False, False, blocking=True)
      $ 1336 "Direction: Base Z+"
      global move_thread_flag_1336=0
      thread move_thread_1336():
        enter_critical
        move_thread_flag_1336 = 1
        local towardsPos=calculate_point_to_move_towards(p[0.0,0.0,0.0,0.0,0.0,0.0], [0.0,0.0,1.0], 0.001)
        movel(towardsPos, a=0.005, v=0.003)
        move_thread_flag_1336 = 2
        exit_critical
      end
      move_thread_flag_1336 = 0
      move_thread_han_1336 = run move_thread_1336()
      while (True):
        sleep(1.0E-10)
        if (move_thread_flag_1336 > 1):
          join move_thread_han_1336
          $ 1337 "Until (distance)"
          break
        end
        sync()
      end
      $ 1338 "Wait: 0.3"
      sleep(0.3)
      $ 1339 "Set CO[1]=Encender"
      set_configurable_digital_out(1, True)
      $ 1340 "Wait: 0.3"
      sleep(0.3)
      $ 1341 "Loop 1 times"
      Loop_54 = 0
      while (Loop_54 < 1):
        $ 1342 "bajar≔pose_add(get_actual_tcp_pose(), bajada_broca)"
        global bajar= pose_add ( get_actual_tcp_pose (), bajada_broca)
        $ 1343 "bajar" "breakAfter"
        movel(bajar, a=0.005, v=0.001)
        $ 1344 "subir≔pose_sub(get_actual_tcp_pose(), bajada_broca)"
        global subir= pose_sub ( get_actual_tcp_pose (), bajada_broca)
        $ 1345 "subir" "breakAfter"
        movel(subir, a=0.01, v=0.01)
        $ 1346 "bajada_broca≔pose_sub(bajada_broca, bajada)"
        global bajada_broca= pose_sub (bajada_broca, bajada)
        Loop_54 = Loop_54 + 1
      end
      $ 1347 "Direction: Base Z+"
      global move_thread_flag_1347=0
      thread move_thread_1347():
        enter_critical
        move_thread_flag_1347 = 1
        local towardsPos=calculate_point_to_move_towards(p[0.0,0.0,0.0,0.0,0.0,0.0], [0.0,0.0,1.0], 0.06)
        movel(towardsPos, a=0.035, v=0.03)
        move_thread_flag_1347 = 2
        exit_critical
      end
      move_thread_flag_1347 = 0
      move_thread_han_1347 = run move_thread_1347()
      while (True):
        sleep(1.0E-10)
        if (move_thread_flag_1347 > 1):
          join move_thread_han_1347
          $ 1348 "Until (distance)"
          break
        end
        sync()
      end
      $ 1349 "Set CO[1]=Apagar"
      set_configurable_digital_out(1, False)
      $ 1350 "barreno_actual≔barreno_actual+1"
      global barreno_actual=barreno_actual+1
      $ 1351 "If barreno_actual≥barrenos_menos1"
      if (barreno_actual >= barrenos_menos1):
        $ 1352 "cambiar_broca≔ True "
        global cambiar_broca=  True
      end
    end
    $ 1355 "Popup: Linea4 con full Terminada!"
    popup("Linea4 con full Terminada!", "Mensaje", False, False, blocking=True)
    $ 1356 "720"
    $ 1357 "Broca_1"
    $ 1358 "Linea5"
    $ 1359 "Marcar_puntos"
    $ 1360 "MoveL"
    $ 1361 "Home3" "breakAfter"
    movel(Home3_p, a=0.5, v=0.1)
    $ 1362 "Linea5_A" "breakAfter"
    movel(Linea5_A_p, a=0.5, v=0.1)
    $ 1363 "Linea5_B" "breakAfter"
    movel(Linea5_B_p, a=0.5, v=0.1)
    $ 1364 "AB"
    $ 1365 "'desbaste_inicial'"
    # 'desbaste_inicial'
    $ 1366 "bajada_broca≔p[0,0,-0.008,0,0,0]"
    global bajada_broca=p[0,0,-0.008,0,0,0]
    $ 1367 "barrenos_menos1≔19"
    global barrenos_menos1=19
    $ 1368 "barreno_actual≔0"
    global barreno_actual=0
    $ 1369 "Loop barreno_actual≤barrenos_menos1"
    while (barreno_actual <= barrenos_menos1):
      $ 1370 "Perforacion"
      $ 1371 "MoveL"
      $ 1372 "internos≔interpolate_pose(Linea5_A, Linea5_B, barreno_actual/barrenos_menos1)"
      global internos= interpolate_pose (Linea5_A_p, Linea5_B_p, barreno_actual/barrenos_menos1)
      $ 1373 "internos" "breakAfter"
      movel(internos, a=0.5, v=0.1)
      $ 1374 "'desbaste_inicial'"
      # 'desbaste_inicial'
      $ 1375 "bajada_broca≔p[0,0,-0.008,0,0,0]"
      global bajada_broca=p[0,0,-0.008,0,0,0]
      $ 1376 "bajada≔p[0,0,0.008,0,0,0]"
      global bajada=p[0,0,0.008,0,0,0]
      $ 1377 "Direction: Base Z-"
      global move_thread_flag_1377=0
      thread move_thread_1377():
        enter_critical
        move_thread_flag_1377 = 1
        local towardsPos=calculate_point_to_move_towards(p[0.0,0.0,0.0,0.0,0.0,0.0], [0.0,0.0,-1.0], 1000.0)
        movel(towardsPos, a=0.005, v=0.007)
        move_thread_flag_1377 = 2
        exit_critical
      end
      move_thread_flag_1377 = 0
      move_thread_han_1377 = run move_thread_1377()
      while (True):
        local targetTcpDirection=get_target_tcp_speed()
        local stepsToRetract=tool_contact(direction=targetTcpDirection)
        if (stepsToRetract > 0):
          kill move_thread_han_1377
          stopl(0.001)
          local backTrackMovement=get_actual_joint_positions_history(stepsToRetract)
          local contactPose=get_forward_kin(backTrackMovement)
          local posDir=[targetTcpDirection[0],targetTcpDirection[1],targetTcpDirection[2]]
          local retractTo=contactPose
          if (norm(posDir) > 1e-6):
            local normalizedPosDir=normalize(posDir)
            local additionalRetraction=p[normalizedPosDir[0] * 0.0, normalizedPosDir[1] * 0.0, normalizedPosDir[2] * 0.0, 0, 0, 0]
            retractTo = pose_sub(contactPose, additionalRetraction)
          end
          movel(retractTo, a=0.001, v=0.1)
          $ 1378 "Until (tool_contact_detection)"
          break
        end
        sync()
      end
      $ 1379 "Popup: punto contacto alanzdo"
      popup("punto contacto alanzdo", "Mensaje", False, False, blocking=True)
      $ 1391 "Direction: Base Z+"
      global move_thread_flag_1391=0
      thread move_thread_1391():
        enter_critical
        move_thread_flag_1391 = 1
        local towardsPos=calculate_point_to_move_towards(p[0.0,0.0,0.0,0.0,0.0,0.0], [0.0,0.0,1.0], 0.15)
        movel(towardsPos, a=0.035, v=0.03)
        move_thread_flag_1391 = 2
        exit_critical
      end
      move_thread_flag_1391 = 0
      move_thread_han_1391 = run move_thread_1391()
      while (True):
        sleep(1.0E-10)
        if (move_thread_flag_1391 > 1):
          join move_thread_han_1391
          $ 1392 "Until (distance)"
          break
        end
        sync()
      end
      $ 1393 "Set CO[1]=Apagar"
      set_configurable_digital_out(1, False)
      $ 1394 "barreno_actual≔barreno_actual+1"
      global barreno_actual=barreno_actual+1
    end
    $ 1463 "Popup: Linea5 con chica Terminada!"
    popup("Linea5 con chica Terminada!", "Mensaje", False, False, blocking=True)
    $ 1464 "Linea6"
    $ 1465 "Marcar_puntos"
    $ 1466 "MoveL"
    $ 1467 "Home3" "breakAfter"
    movel(Home3_p, a=0.5, v=0.1)
    $ 1468 "Linea4_A" "breakAfter"
    movel(Linea4_A_p, a=0.5, v=0.1)
    $ 1469 "Linea4_B" "breakAfter"
    movel(Linea4_B_p, a=0.5, v=0.1)
    $ 1470 "Linea4_C" "breakAfter"
    movel(Linea4_C_p, a=0.5, v=0.1)
    $ 1471 "Linea4_D" "breakAfter"
    movel(Linea4_D_p, a=0.5, v=0.1)
    $ 1472 "Linea4_E" "breakAfter"
    movel(Linea4_E_p, a=0.5, v=0.1)
    $ 1473 "Linea4_F" "breakAfter"
    movel(Linea4_F_p, a=0.5, v=0.1)
    $ 1474 "AB"
    $ 1475 "'desbaste_inicial'"
    # 'desbaste_inicial'
    $ 1476 "bajada_broca≔p[0,0,-0.008,0,0,0]"
    global bajada_broca=p[0,0,-0.008,0,0,0]
    $ 1477 "barrenos_menos1≔8"
    global barrenos_menos1=8
    $ 1478 "barreno_actual≔0"
    global barreno_actual=0
    $ 1479 "Loop barreno_actual≤barrenos_menos1"
    while (barreno_actual <= barrenos_menos1):
      $ 1480 "Perforacion"
      $ 1481 "MoveL"
      $ 1482 "internos≔interpolate_pose(Linea4_A, Linea4_B, barreno_actual/barrenos_menos1)"
      global internos= interpolate_pose (Linea4_A_p, Linea4_B_p, barreno_actual/barrenos_menos1)
      $ 1483 "internos" "breakAfter"
      movel(internos, a=0.5, v=0.1)
      $ 1484 "'desbaste_inicial'"
      # 'desbaste_inicial'
      $ 1485 "bajada_broca≔p[0,0,-0.008,0,0,0]"
      global bajada_broca=p[0,0,-0.008,0,0,0]
      $ 1486 "bajada≔p[0,0,0.008,0,0,0]"
      global bajada=p[0,0,0.008,0,0,0]
      $ 1487 "Direction: Base Z-"
      global move_thread_flag_1487=0
      thread move_thread_1487():
        enter_critical
        move_thread_flag_1487 = 1
        local towardsPos=calculate_point_to_move_towards(p[0.0,0.0,0.0,0.0,0.0,0.0], [0.0,0.0,-1.0], 0.055)
        movel(towardsPos, a=0.015, v=0.02)
        move_thread_flag_1487 = 2
        exit_critical
      end
      move_thread_flag_1487 = 0
      move_thread_han_1487 = run move_thread_1487()
      while (True):
        sleep(1.0E-10)
        if (move_thread_flag_1487 > 1):
          join move_thread_han_1487
          $ 1488 "Until (distance)"
          break
        end
        sync()
      end
      $ 1489 "Popup: punto contacto alanzdo"
      popup("punto contacto alanzdo", "Mensaje", False, False, blocking=True)
      $ 1490 "Direction: Base Z+"
      global move_thread_flag_1490=0
      thread move_thread_1490():
        enter_critical
        move_thread_flag_1490 = 1
        local towardsPos=calculate_point_to_move_towards(p[0.0,0.0,0.0,0.0,0.0,0.0], [0.0,0.0,1.0], 0.002)
        movel(towardsPos, a=0.005, v=0.003)
        move_thread_flag_1490 = 2
        exit_critical
      end
      move_thread_flag_1490 = 0
      move_thread_han_1490 = run move_thread_1490()
      while (True):
        sleep(1.0E-10)
        if (move_thread_flag_1490 > 1):
          join move_thread_han_1490
          $ 1491 "Until (distance)"
          break
        end
        sync()
      end
      $ 1492 "Wait: 0.3"
      sleep(0.3)
      $ 1493 "Set CO[1]=Encender"
      set_configurable_digital_out(1, True)
      $ 1494 "Wait: 0.3"
      sleep(0.3)
      $ 1495 "Loop 3 times"
      Loop_61 = 0
      while (Loop_61 < 3):
        $ 1496 "bajar≔pose_add(get_actual_tcp_pose(), bajada_broca)"
        global bajar= pose_add ( get_actual_tcp_pose (), bajada_broca)
        $ 1497 "bajar" "breakAfter"
        movel(bajar, a=0.005, v=0.001)
        $ 1498 "subir≔pose_sub(get_actual_tcp_pose(), bajada_broca)"
        global subir= pose_sub ( get_actual_tcp_pose (), bajada_broca)
        $ 1499 "subir" "breakAfter"
        movel(subir, a=0.01, v=0.01)
        $ 1500 "bajada_broca≔pose_sub(bajada_broca, bajada)"
        global bajada_broca= pose_sub (bajada_broca, bajada)
        Loop_61 = Loop_61 + 1
      end
      $ 1501 "Direction: Base Z+"
      global move_thread_flag_1501=0
      thread move_thread_1501():
        enter_critical
        move_thread_flag_1501 = 1
        local towardsPos=calculate_point_to_move_towards(p[0.0,0.0,0.0,0.0,0.0,0.0], [0.0,0.0,1.0], 0.06)
        movel(towardsPos, a=0.035, v=0.03)
        move_thread_flag_1501 = 2
        exit_critical
      end
      move_thread_flag_1501 = 0
      move_thread_han_1501 = run move_thread_1501()
      while (True):
        sleep(1.0E-10)
        if (move_thread_flag_1501 > 1):
          join move_thread_han_1501
          $ 1502 "Until (distance)"
          break
        end
        sync()
      end
      $ 1503 "Set CO[1]=Apagar"
      set_configurable_digital_out(1, False)
      $ 1504 "barreno_actual≔barreno_actual+1"
      global barreno_actual=barreno_actual+1
    end
    $ 1507 "CD"
    $ 1508 "'desbaste_inicial'"
    # 'desbaste_inicial'
    $ 1509 "bajada_broca≔p[0,0,-0.008,0,0,0]"
    global bajada_broca=p[0,0,-0.008,0,0,0]
    $ 1510 "barrenos_menos1≔8"
    global barrenos_menos1=8
    $ 1511 "barreno_actual≔0"
    global barreno_actual=0
    $ 1512 "Loop barreno_actual≤barrenos_menos1"
    while (barreno_actual <= barrenos_menos1):
      $ 1513 "Perforacion"
      $ 1514 "MoveL"
      $ 1515 "internos≔interpolate_pose(Linea4_C, Linea4_D, barreno_actual/barrenos_menos1)"
      global internos= interpolate_pose (Linea4_C_p, Linea4_D_p, barreno_actual/barrenos_menos1)
      $ 1516 "internos" "breakAfter"
      movel(internos, a=0.5, v=0.1)
      $ 1517 "'desbaste_inicial'"
      # 'desbaste_inicial'
      $ 1518 "bajada_broca≔p[0,0,-0.008,0,0,0]"
      global bajada_broca=p[0,0,-0.008,0,0,0]
      $ 1519 "bajada≔p[0,0,0.008,0,0,0]"
      global bajada=p[0,0,0.008,0,0,0]
      $ 1520 "Direction: Base Z-"
      global move_thread_flag_1520=0
      thread move_thread_1520():
        enter_critical
        move_thread_flag_1520 = 1
        local towardsPos=calculate_point_to_move_towards(p[0.0,0.0,0.0,0.0,0.0,0.0], [0.0,0.0,-1.0], 0.055)
        movel(towardsPos, a=0.015, v=0.02)
        move_thread_flag_1520 = 2
        exit_critical
      end
      move_thread_flag_1520 = 0
      move_thread_han_1520 = run move_thread_1520()
      while (True):
        sleep(1.0E-10)
        if (move_thread_flag_1520 > 1):
          join move_thread_han_1520
          $ 1521 "Until (distance)"
          break
        end
        sync()
      end
      $ 1522 "Popup: punto contacto alanzdo"
      popup("punto contacto alanzdo", "Mensaje", False, False, blocking=True)
      $ 1523 "Direction: Base Z+"
      global move_thread_flag_1523=0
      thread move_thread_1523():
        enter_critical
        move_thread_flag_1523 = 1
        local towardsPos=calculate_point_to_move_towards(p[0.0,0.0,0.0,0.0,0.0,0.0], [0.0,0.0,1.0], 0.002)
        movel(towardsPos, a=0.005, v=0.003)
        move_thread_flag_1523 = 2
        exit_critical
      end
      move_thread_flag_1523 = 0
      move_thread_han_1523 = run move_thread_1523()
      while (True):
        sleep(1.0E-10)
        if (move_thread_flag_1523 > 1):
          join move_thread_han_1523
          $ 1524 "Until (distance)"
          break
        end
        sync()
      end
      $ 1525 "Wait: 0.3"
      sleep(0.3)
      $ 1526 "Set CO[1]=Encender"
      set_configurable_digital_out(1, True)
      $ 1527 "Wait: 0.3"
      sleep(0.3)
      $ 1528 "Loop 3 times"
      Loop_63 = 0
      while (Loop_63 < 3):
        $ 1529 "bajar≔pose_add(get_actual_tcp_pose(), bajada_broca)"
        global bajar= pose_add ( get_actual_tcp_pose (), bajada_broca)
        $ 1530 "bajar" "breakAfter"
        movel(bajar, a=0.005, v=0.001)
        $ 1531 "subir≔pose_sub(get_actual_tcp_pose(), bajada_broca)"
        global subir= pose_sub ( get_actual_tcp_pose (), bajada_broca)
        $ 1532 "subir" "breakAfter"
        movel(subir, a=0.01, v=0.01)
        $ 1533 "bajada_broca≔pose_sub(bajada_broca, bajada)"
        global bajada_broca= pose_sub (bajada_broca, bajada)
        Loop_63 = Loop_63 + 1
      end
      $ 1534 "Direction: Base Z+"
      global move_thread_flag_1534=0
      thread move_thread_1534():
        enter_critical
        move_thread_flag_1534 = 1
        local towardsPos=calculate_point_to_move_towards(p[0.0,0.0,0.0,0.0,0.0,0.0], [0.0,0.0,1.0], 0.06)
        movel(towardsPos, a=0.035, v=0.03)
        move_thread_flag_1534 = 2
        exit_critical
      end
      move_thread_flag_1534 = 0
      move_thread_han_1534 = run move_thread_1534()
      while (True):
        sleep(1.0E-10)
        if (move_thread_flag_1534 > 1):
          join move_thread_han_1534
          $ 1535 "Until (distance)"
          break
        end
        sync()
      end
      $ 1536 "Set CO[1]=Apagar"
      set_configurable_digital_out(1, False)
      $ 1537 "barreno_actual≔barreno_actual+1"
      global barreno_actual=barreno_actual+1
    end
    $ 1540 "EF"
    $ 1541 "'desbaste_inicial'"
    # 'desbaste_inicial'
    $ 1542 "bajada_broca≔p[0,0,-0.008,0,0,0]"
    global bajada_broca=p[0,0,-0.008,0,0,0]
    $ 1543 "barrenos_menos1≔8"
    global barrenos_menos1=8
    $ 1544 "barreno_actual≔0"
    global barreno_actual=0
    $ 1545 "Loop barreno_actual≤barrenos_menos1"
    while (barreno_actual <= barrenos_menos1):
      $ 1546 "Perforacion"
      $ 1547 "MoveL"
      $ 1548 "internos≔interpolate_pose(Linea4_E, Linea4_F, barreno_actual/barrenos_menos1)"
      global internos= interpolate_pose (Linea4_E_p, Linea4_F_p, barreno_actual/barrenos_menos1)
      $ 1549 "internos" "breakAfter"
      movel(internos, a=0.5, v=0.1)
      $ 1550 "'desbaste_inicial'"
      # 'desbaste_inicial'
      $ 1551 "bajada_broca≔p[0,0,-0.008,0,0,0]"
      global bajada_broca=p[0,0,-0.008,0,0,0]
      $ 1552 "bajada≔p[0,0,0.008,0,0,0]"
      global bajada=p[0,0,0.008,0,0,0]
      $ 1553 "Direction: Base Z-"
      global move_thread_flag_1553=0
      thread move_thread_1553():
        enter_critical
        move_thread_flag_1553 = 1
        local towardsPos=calculate_point_to_move_towards(p[0.0,0.0,0.0,0.0,0.0,0.0], [0.0,0.0,-1.0], 0.055)
        movel(towardsPos, a=0.015, v=0.02)
        move_thread_flag_1553 = 2
        exit_critical
      end
      move_thread_flag_1553 = 0
      move_thread_han_1553 = run move_thread_1553()
      while (True):
        sleep(1.0E-10)
        if (move_thread_flag_1553 > 1):
          join move_thread_han_1553
          $ 1554 "Until (distance)"
          break
        end
        sync()
      end
      $ 1555 "Popup: punto contacto alanzdo"
      popup("punto contacto alanzdo", "Mensaje", False, False, blocking=True)
      $ 1556 "Direction: Base Z+"
      global move_thread_flag_1556=0
      thread move_thread_1556():
        enter_critical
        move_thread_flag_1556 = 1
        local towardsPos=calculate_point_to_move_towards(p[0.0,0.0,0.0,0.0,0.0,0.0], [0.0,0.0,1.0], 0.002)
        movel(towardsPos, a=0.005, v=0.003)
        move_thread_flag_1556 = 2
        exit_critical
      end
      move_thread_flag_1556 = 0
      move_thread_han_1556 = run move_thread_1556()
      while (True):
        sleep(1.0E-10)
        if (move_thread_flag_1556 > 1):
          join move_thread_han_1556
          $ 1557 "Until (distance)"
          break
        end
        sync()
      end
      $ 1558 "Wait: 0.3"
      sleep(0.3)
      $ 1559 "Set CO[1]=Encender"
      set_configurable_digital_out(1, True)
      $ 1560 "Wait: 0.3"
      sleep(0.3)
      $ 1561 "Loop 3 times"
      Loop_65 = 0
      while (Loop_65 < 3):
        $ 1562 "bajar≔pose_add(get_actual_tcp_pose(), bajada_broca)"
        global bajar= pose_add ( get_actual_tcp_pose (), bajada_broca)
        $ 1563 "bajar" "breakAfter"
        movel(bajar, a=0.005, v=0.001)
        $ 1564 "subir≔pose_sub(get_actual_tcp_pose(), bajada_broca)"
        global subir= pose_sub ( get_actual_tcp_pose (), bajada_broca)
        $ 1565 "subir" "breakAfter"
        movel(subir, a=0.01, v=0.01)
        $ 1566 "bajada_broca≔pose_sub(bajada_broca, bajada)"
        global bajada_broca= pose_sub (bajada_broca, bajada)
        Loop_65 = Loop_65 + 1
      end
      $ 1567 "Direction: Base Z+"
      global move_thread_flag_1567=0
      thread move_thread_1567():
        enter_critical
        move_thread_flag_1567 = 1
        local towardsPos=calculate_point_to_move_towards(p[0.0,0.0,0.0,0.0,0.0,0.0], [0.0,0.0,1.0], 0.06)
        movel(towardsPos, a=0.035, v=0.03)
        move_thread_flag_1567 = 2
        exit_critical
      end
      move_thread_flag_1567 = 0
      move_thread_han_1567 = run move_thread_1567()
      while (True):
        sleep(1.0E-10)
        if (move_thread_flag_1567 > 1):
          join move_thread_han_1567
          $ 1568 "Until (distance)"
          break
        end
        sync()
      end
      $ 1569 "Set CO[1]=Apagar"
      set_configurable_digital_out(1, False)
      $ 1570 "barreno_actual≔barreno_actual+1"
      global barreno_actual=barreno_actual+1
      $ 1571 "If barreno_actual≥barrenos_menos1"
      if (barreno_actual >= barrenos_menos1):
        $ 1572 "cambiar_broca≔ True "
        global cambiar_broca=  True
      end
    end
    $ 1575 "Popup: Linea6 con chica Terminada!"
    popup("Linea6 con chica Terminada!", "Mensaje", False, False, blocking=True)
    $ 1576 "'Subprogramas:'"
    # 'Subprogramas:'
  end
end
